Yaskawa INFORM job: A_ROOF_SIDE_0617_2_PAINT_46.JBI

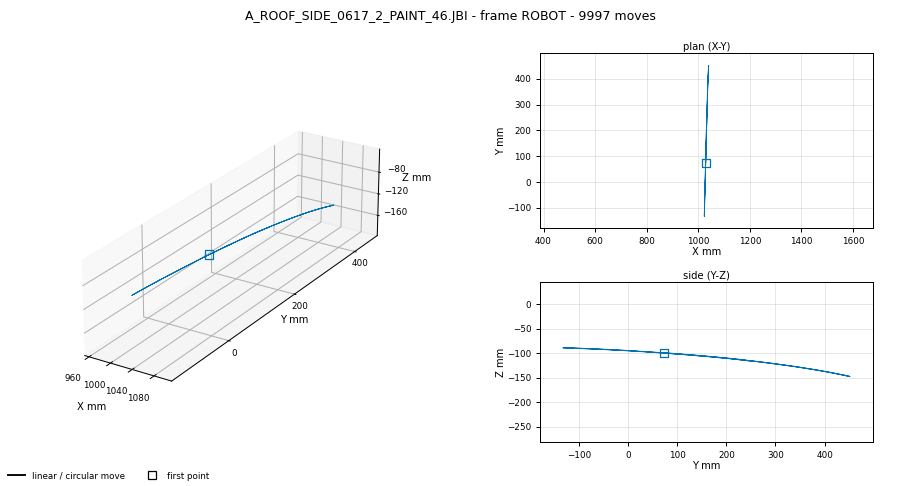
[picture p0: tool path of A_ROOF_SIDE_0617_2_PAINT_46.JBI in frame ROBOT, 9997 of 9997 moves have a stored position in this frame; points joined in program order, loops and branches not executed]
/JOB
//NAME A_ROOF_SIDE_0617_2_PAINT46
//POS
///NPOS 9997,0,0,0,0,0
///TOOL 1
///USER 0
///POSTYPE ROBOT
///RECTAN
///RCONF 1,0,0,0,0,0,0,0,0,0,0,0,0,0,0,0,0,0,0,0,0,0,0,0
C00000=1029.053,72.292,-98.591,168.354,44.972,158.390
C00001=1029.059,72.542,-98.608,168.356,44.969,158.390
C00002=1029.064,72.791,-98.626,168.358,44.967,158.389
C00003=1029.071,73.040,-98.644,168.360,44.965,158.389
C00004=1029.078,73.289,-98.662,168.362,44.963,158.389
C00005=1029.083,73.538,-98.680,168.365,44.961,158.389
C00006=1029.089,73.788,-98.698,168.367,44.958,158.389
C00007=1029.095,74.038,-98.715,168.370,44.956,158.388
C00008=1029.101,74.286,-98.734,168.373,44.954,158.388
C00009=1029.108,74.536,-98.751,168.375,44.951,158.388
C00010=1029.114,74.785,-98.769,168.377,44.949,158.388
C00011=1029.119,75.016,-98.786,168.380,44.947,158.388
C00012=1029.126,75.246,-98.802,168.381,44.945,158.387
C00013=1029.131,75.476,-98.818,168.384,44.943,158.387
C00014=1029.136,75.706,-98.836,168.386,44.941,158.387
C00015=1029.143,75.937,-98.852,168.389,44.939,158.387
C00016=1029.148,76.166,-98.868,168.390,44.937,158.387
C00017=1029.154,76.397,-98.886,168.393,44.935,158.387
C00018=1029.160,76.627,-98.902,168.395,44.933,158.387
C00019=1029.166,76.877,-98.920,168.398,44.931,158.386
C00020=1029.172,77.126,-98.938,168.400,44.928,158.386
C00021=1029.178,77.375,-98.956,168.403,44.926,158.386
C00022=1029.184,77.624,-98.974,168.405,44.924,158.386
C00023=1029.190,77.874,-98.992,168.408,44.922,158.386
C00024=1029.196,78.123,-99.010,168.409,44.920,158.385
C00025=1029.202,78.372,-99.029,168.412,44.917,158.385
C00026=1029.208,78.622,-99.047,168.414,44.915,158.385
C00027=1029.215,78.871,-99.065,168.417,44.913,158.385
C00028=1029.220,79.120,-99.083,168.419,44.911,158.385
C00029=1029.227,79.369,-99.101,168.422,44.909,158.385
C00030=1029.233,79.619,-99.119,168.424,44.907,158.384
C00031=1029.238,79.868,-99.138,168.427,44.905,158.384
C00032=1029.244,80.118,-99.156,168.429,44.902,158.384
C00033=1029.250,80.367,-99.175,168.432,44.900,158.384
C00034=1029.257,80.616,-99.193,168.434,44.898,158.384
C00035=1029.262,80.865,-99.211,168.437,44.895,158.383
C00036=1029.269,81.114,-99.230,168.438,44.894,158.383
C00037=1029.275,81.364,-99.248,168.441,44.892,158.383
C00038=1029.281,81.613,-99.266,168.443,44.889,158.383
C00039=1029.288,81.863,-99.284,168.446,44.887,158.383
C00040=1029.293,82.111,-99.302,168.448,44.885,158.383
C00041=1029.299,82.361,-99.320,168.450,44.883,158.382
C00042=1029.305,82.610,-99.340,168.453,44.881,158.382
C00043=1029.312,82.859,-99.358,168.456,44.879,158.382
C00044=1029.317,83.108,-99.376,168.458,44.876,158.382
C00045=1029.324,83.357,-99.395,168.460,44.874,158.382
C00046=1029.330,83.607,-99.412,168.463,44.872,158.382
C00047=1029.336,83.856,-99.431,168.465,44.869,158.381
C00048=1029.343,84.105,-99.450,168.468,44.867,158.381
C00049=1029.348,84.354,-99.467,168.470,44.865,158.381
C00050=1029.354,84.604,-99.486,168.473,44.863,158.381
C00051=1029.361,84.853,-99.505,168.475,44.861,158.381
C00052=1029.366,85.103,-99.523,168.477,44.858,158.380
C00053=1029.373,85.352,-99.542,168.479,44.856,158.380
C00054=1029.379,85.601,-99.560,168.482,44.855,158.380
C00055=1029.385,85.850,-99.578,168.484,44.852,158.380
C00056=1029.391,86.099,-99.597,168.487,44.850,158.380
C00057=1029.397,86.348,-99.615,168.489,44.847,158.379
C00058=1029.404,86.598,-99.633,168.492,44.845,158.379
C00059=1029.410,86.847,-99.652,168.494,44.843,158.379
C00060=1029.416,87.096,-99.671,168.496,44.841,158.379
C00061=1029.422,87.346,-99.690,168.499,44.839,158.379
C00062=1029.428,87.595,-99.707,168.501,44.836,158.378
C00063=1029.434,87.844,-99.726,168.504,44.834,158.378
C00064=1029.441,88.093,-99.745,168.506,44.832,158.378
C00065=1029.447,88.343,-99.763,168.509,44.830,158.378
C00066=1029.453,88.592,-99.781,168.511,44.828,158.378
C00067=1029.459,88.841,-99.800,168.514,44.825,158.378
C00068=1029.466,89.090,-99.819,168.516,44.823,158.377
C00069=1029.472,89.340,-99.838,168.519,44.820,158.377
C00070=1029.478,89.589,-99.856,168.521,44.818,158.377
C00071=1029.484,89.838,-99.874,168.524,44.816,158.377
C00072=1029.490,90.087,-99.893,168.526,44.814,158.377
C00073=1029.496,90.336,-99.912,168.529,44.812,158.376
C00074=1029.502,90.585,-99.931,168.531,44.810,158.376
C00075=1029.508,90.835,-99.950,168.533,44.807,158.376
C00076=1029.514,91.084,-99.968,168.535,44.806,158.376
C00077=1029.520,91.334,-99.987,168.538,44.804,158.376
C00078=1029.526,91.583,-100.006,168.540,44.802,158.376
C00079=1029.533,91.868,-100.028,168.544,44.799,158.375
C00080=1029.540,92.153,-100.049,168.546,44.796,158.375
C00081=1029.547,92.438,-100.070,168.548,44.794,158.375
C00082=1029.554,92.723,-100.092,168.552,44.791,158.375
C00083=1029.560,92.973,-100.111,168.554,44.789,158.375
C00084=1029.566,93.222,-100.130,168.557,44.787,158.375
C00085=1029.572,93.470,-100.148,168.559,44.785,158.374
C00086=1029.578,93.720,-100.167,168.561,44.783,158.374
C00087=1029.584,93.969,-100.186,168.563,44.781,158.374
C00088=1029.590,94.218,-100.205,168.566,44.779,158.374
C00089=1029.596,94.467,-100.224,168.568,44.777,158.374
C00090=1029.602,94.717,-100.243,168.571,44.775,158.373
C00091=1029.608,94.966,-100.262,168.573,44.772,158.373
C00092=1029.615,95.215,-100.281,168.576,44.770,158.373
C00093=1029.621,95.464,-100.299,168.578,44.768,158.373
C00094=1029.627,95.714,-100.319,168.581,44.765,158.373
C00095=1029.633,95.963,-100.337,168.583,44.763,158.372
C00096=1029.639,96.212,-100.356,168.586,44.762,158.372
C00097=1029.645,96.461,-100.375,168.588,44.759,158.372
C00098=1029.651,96.711,-100.394,168.591,44.757,158.372
C00099=1029.657,96.960,-100.413,168.593,44.755,158.372
C00100=1029.664,97.209,-100.432,168.596,44.752,158.371
C00101=1029.669,97.459,-100.451,168.598,44.750,158.371
C00102=1029.676,97.707,-100.470,168.601,44.748,158.371
C00103=1029.682,97.956,-100.490,168.603,44.746,158.371
C00104=1029.688,98.206,-100.508,168.606,44.744,158.371
C00105=1029.694,98.455,-100.527,168.608,44.741,158.371
C00106=1029.700,98.704,-100.546,168.610,44.739,158.370
C00107=1029.706,98.954,-100.565,168.613,44.737,158.370
C00108=1029.712,99.203,-100.584,168.615,44.735,158.370
C00109=1029.719,99.452,-100.603,168.618,44.733,158.370
C00110=1029.725,99.701,-100.623,168.620,44.731,158.370
C00111=1029.731,99.950,-100.641,168.623,44.728,158.369
C00112=1029.737,100.199,-100.660,168.625,44.726,158.369
C00113=1029.743,100.449,-100.680,168.628,44.724,158.369
C00114=1029.748,100.698,-100.699,168.631,44.722,158.369
C00115=1029.755,100.947,-100.718,168.632,44.720,158.369
C00116=1029.761,101.196,-100.738,168.634,44.718,158.369
C00117=1029.766,101.445,-100.757,168.637,44.716,158.368
C00118=1029.773,101.694,-100.776,168.640,44.714,158.368
C00119=1029.779,101.943,-100.795,168.642,44.711,158.368
C00120=1029.785,102.193,-100.815,168.644,44.710,158.368
C00121=1029.791,102.442,-100.835,168.647,44.708,158.368
C00122=1029.798,102.691,-100.854,168.650,44.706,158.368
C00123=1029.803,102.941,-100.873,168.652,44.703,158.367
C00124=1029.809,103.190,-100.893,168.654,44.701,158.367
C00125=1029.816,103.439,-100.911,168.657,44.699,158.367
C00126=1029.821,103.688,-100.931,168.660,44.697,158.367
C00127=1029.827,103.937,-100.951,168.662,44.695,158.367
C00128=1029.833,104.186,-100.970,168.665,44.693,158.367
C00129=1029.840,104.436,-100.989,168.667,44.691,158.366
C00130=1029.846,104.684,-101.009,168.670,44.689,158.366
C00131=1029.851,104.934,-101.028,168.672,44.686,158.366
C00132=1029.857,105.183,-101.047,168.675,44.684,158.366
C00133=1029.864,105.432,-101.066,168.677,44.682,158.366
C00134=1029.870,105.682,-101.086,168.679,44.680,158.365
C00135=1029.876,105.931,-101.106,168.682,44.678,158.365
C00136=1029.882,106.180,-101.125,168.685,44.676,158.365
C00137=1029.888,106.429,-101.145,168.687,44.674,158.365
C00138=1029.894,106.678,-101.164,168.690,44.671,158.365
C00139=1029.900,106.928,-101.183,168.692,44.669,158.365
C00140=1029.906,107.176,-101.202,168.695,44.667,158.365
C00141=1029.912,107.425,-101.222,168.697,44.665,158.364
C00142=1029.919,107.675,-101.242,168.700,44.663,158.364
C00143=1029.926,107.960,-101.264,168.702,44.660,158.364
C00144=1029.932,108.245,-101.286,168.705,44.658,158.364
C00145=1029.939,108.530,-101.308,168.708,44.655,158.363
C00146=1029.947,108.815,-101.331,168.710,44.653,158.363
C00147=1029.953,109.064,-101.350,168.713,44.651,158.363
C00148=1029.959,109.313,-101.370,168.715,44.649,158.363
C00149=1029.964,109.563,-101.389,168.718,44.647,158.363
C00150=1029.971,109.811,-101.409,168.720,44.644,158.363
C00151=1029.977,110.061,-101.428,168.723,44.642,158.362
C00152=1029.983,110.310,-101.448,168.725,44.640,158.362
C00153=1029.989,110.560,-101.468,168.728,44.638,158.362
C00154=1029.995,110.808,-101.488,168.730,44.636,158.362
C00155=1030.001,111.058,-101.507,168.733,44.634,158.362
C00156=1030.007,111.307,-101.527,168.735,44.632,158.362
C00157=1030.013,111.556,-101.547,168.738,44.629,158.361
C00158=1030.020,111.805,-101.566,168.740,44.627,158.361
C00159=1030.026,112.054,-101.586,168.743,44.625,158.361
C00160=1030.032,112.303,-101.606,168.745,44.624,158.361
C00161=1030.038,112.553,-101.625,168.748,44.621,158.361
C00162=1030.044,112.802,-101.645,168.750,44.619,158.360
C00163=1030.050,113.051,-101.665,168.753,44.617,158.360
C00164=1030.056,113.300,-101.684,168.755,44.615,158.360
C00165=1030.061,113.549,-101.705,168.758,44.613,158.360
C00166=1030.068,113.799,-101.725,168.761,44.611,158.360
C00167=1030.074,114.048,-101.745,168.763,44.609,158.360
C00168=1030.079,114.297,-101.764,168.766,44.607,158.360
C00169=1030.085,114.546,-101.784,168.768,44.605,158.359
C00170=1030.091,114.795,-101.804,168.771,44.603,158.359
C00171=1030.097,115.044,-101.825,168.773,44.601,158.359
C00172=1030.103,115.293,-101.845,168.776,44.599,158.359
C00173=1030.109,115.542,-101.865,168.778,44.597,158.359
C00174=1030.115,115.791,-101.884,168.781,44.595,158.359
C00175=1030.121,116.040,-101.904,168.784,44.593,158.359
C00176=1030.127,116.290,-101.925,168.786,44.591,158.358
C00177=1030.133,116.539,-101.945,168.788,44.589,158.358
C00178=1030.139,116.788,-101.965,168.791,44.587,158.358
C00179=1030.145,117.037,-101.985,168.794,44.585,158.358
C00180=1030.151,117.286,-102.006,168.796,44.583,158.358
C00181=1030.156,117.536,-102.025,168.799,44.581,158.358
C00182=1030.162,117.785,-102.045,168.801,44.579,158.357
C00183=1030.168,118.033,-102.065,168.804,44.577,158.357
C00184=1030.175,118.283,-102.086,168.806,44.575,158.357
C00185=1030.181,118.532,-102.106,168.809,44.572,158.357
C00186=1030.186,118.781,-102.126,168.811,44.570,158.357
C00187=1030.192,119.030,-102.146,168.814,44.568,158.357
C00188=1030.199,119.279,-102.166,168.817,44.567,158.357
C00189=1030.205,119.528,-102.186,168.819,44.565,158.356
C00190=1030.210,119.777,-102.207,168.822,44.563,158.356
C00191=1030.216,120.027,-102.227,168.824,44.561,158.356
C00192=1030.222,120.275,-102.247,168.827,44.558,158.356
C00193=1030.228,120.524,-102.267,168.829,44.556,158.356
C00194=1030.234,120.773,-102.287,168.832,44.554,158.356
C00195=1030.240,121.023,-102.308,168.834,44.552,158.355
C00196=1030.246,121.272,-102.328,168.837,44.550,158.355
C00197=1030.252,121.521,-102.348,168.839,44.548,158.355
C00198=1030.259,121.770,-102.368,168.842,44.546,158.355
C00199=1030.264,122.019,-102.389,168.844,44.544,158.355
C00200=1030.270,122.268,-102.409,168.847,44.542,158.355
C00201=1030.277,122.518,-102.429,168.849,44.540,158.354
C00202=1030.283,122.766,-102.449,168.852,44.538,158.354
C00203=1030.289,123.015,-102.469,168.855,44.536,158.354
C00204=1030.295,123.265,-102.490,168.857,44.534,158.354
C00205=1030.300,123.514,-102.510,168.860,44.532,158.354
C00206=1030.307,123.763,-102.530,168.862,44.530,158.354
C00207=1030.313,124.048,-102.554,168.865,44.527,158.353
C00208=1030.321,124.333,-102.577,168.868,44.525,158.353
C00209=1030.328,124.618,-102.600,168.871,44.522,158.353
C00210=1030.335,124.903,-102.624,168.874,44.520,158.353
C00211=1030.341,125.152,-102.644,168.877,44.518,158.353
C00212=1030.347,125.401,-102.663,168.879,44.516,158.353
C00213=1030.353,125.650,-102.684,168.881,44.514,158.352
C00214=1030.359,125.899,-102.704,168.885,44.512,158.352
C00215=1030.365,126.149,-102.725,168.888,44.510,158.352
C00216=1030.371,126.398,-102.745,168.890,44.508,158.352
C00217=1030.378,126.647,-102.766,168.893,44.506,158.352
C00218=1030.383,126.896,-102.786,168.895,44.503,158.352
C00219=1030.389,127.145,-102.806,168.898,44.501,158.351
C00220=1030.396,127.394,-102.827,168.900,44.499,158.351
C00221=1030.402,127.643,-102.846,168.903,44.497,158.351
C00222=1030.408,127.893,-102.867,168.905,44.496,158.351
C00223=1030.414,128.141,-102.888,168.908,44.493,158.351
C00224=1030.421,128.390,-102.908,168.910,44.491,158.351
C00225=1030.427,128.639,-102.928,168.913,44.489,158.350
C00226=1030.432,128.889,-102.949,168.916,44.487,158.350
C00227=1030.439,129.137,-102.970,168.919,44.485,158.350
C00228=1030.445,129.387,-102.990,168.921,44.482,158.350
C00229=1030.451,129.636,-103.010,168.924,44.481,158.350
C00230=1030.457,129.885,-103.031,168.927,44.479,158.350
C00231=1030.463,130.134,-103.051,168.929,44.477,158.350
C00232=1030.470,130.383,-103.072,168.931,44.474,158.349
C00233=1030.475,130.632,-103.093,168.934,44.472,158.349
C00234=1030.482,130.882,-103.113,168.937,44.470,158.349
C00235=1030.487,131.130,-103.134,168.939,44.468,158.349
C00236=1030.493,131.379,-103.154,168.942,44.466,158.349
C00237=1030.500,131.628,-103.176,168.945,44.464,158.349
C00238=1030.506,131.877,-103.196,168.948,44.462,158.348
C00239=1030.511,132.127,-103.217,168.951,44.460,158.348
C00240=1030.517,132.375,-103.238,168.953,44.458,158.348
C00241=1030.524,132.625,-103.258,168.956,44.457,158.348
C00242=1030.529,132.873,-103.280,168.958,44.455,158.348
C00243=1030.536,133.123,-103.300,168.961,44.453,158.348
C00244=1030.541,133.371,-103.321,168.963,44.451,158.348
C00245=1030.547,133.621,-103.342,168.966,44.449,158.347
C00246=1030.554,133.869,-103.363,168.969,44.447,158.347
C00247=1030.559,134.119,-103.384,168.971,44.445,158.347
C00248=1030.566,134.367,-103.404,168.973,44.442,158.347
C00249=1030.572,134.617,-103.425,168.976,44.440,158.347
C00250=1030.578,134.865,-103.446,168.980,44.438,158.347
C00251=1030.584,135.115,-103.467,168.982,44.436,158.347
C00252=1030.589,135.364,-103.488,168.985,44.434,158.346
C00253=1030.596,135.613,-103.509,168.987,44.433,158.346
C00254=1030.602,135.863,-103.530,168.990,44.431,158.346
C00255=1030.608,136.111,-103.550,168.993,44.429,158.346
C00256=1030.614,136.361,-103.572,168.995,44.427,158.346
C00257=1030.619,136.610,-103.592,168.998,44.425,158.346
C00258=1030.626,136.859,-103.613,169.000,44.423,158.346
C00259=1030.632,137.107,-103.635,169.003,44.421,158.345
C00260=1030.638,137.357,-103.656,169.006,44.419,158.345
C00261=1030.644,137.605,-103.676,169.009,44.417,158.345
C00262=1030.650,137.855,-103.697,169.012,44.415,158.345
C00263=1030.656,138.104,-103.719,169.014,44.413,158.345
C00264=1030.662,138.352,-103.739,169.017,44.411,158.345
C00265=1030.668,138.602,-103.760,169.019,44.409,158.345
C00266=1030.674,138.851,-103.782,169.022,44.407,158.344
C00267=1030.680,139.100,-103.803,169.024,44.405,158.344
C00268=1030.686,139.350,-103.824,169.027,44.404,158.344
C00269=1030.692,139.598,-103.845,169.031,44.401,158.344
C00270=1030.698,139.847,-103.867,169.033,44.399,158.344
C00271=1030.705,140.133,-103.891,169.036,44.398,158.344
C00272=1030.711,140.417,-103.915,169.039,44.395,158.344
C00273=1030.719,140.702,-103.939,169.042,44.393,158.343
C00274=1030.725,140.987,-103.964,169.045,44.391,158.343
C00275=1030.731,141.235,-103.985,169.048,44.389,158.343
C00276=1030.737,141.485,-104.006,169.050,44.387,158.343
C00277=1030.743,141.734,-104.027,169.053,44.385,158.343
C00278=1030.749,141.982,-104.049,169.056,44.383,158.343
C00279=1030.755,142.232,-104.070,169.059,44.381,158.343
C00280=1030.761,142.480,-104.092,169.062,44.379,158.343
C00281=1030.767,142.730,-104.112,169.064,44.377,158.342
C00282=1030.774,142.979,-104.133,169.067,44.375,158.342
C00283=1030.779,143.227,-104.155,169.069,44.373,158.342
C00284=1030.785,143.477,-104.176,169.072,44.371,158.342
C00285=1030.791,143.726,-104.198,169.075,44.369,158.342
C00286=1030.797,143.974,-104.219,169.078,44.367,158.342
C00287=1030.803,144.224,-104.240,169.081,44.365,158.342
C00288=1030.809,144.473,-104.262,169.083,44.363,158.341
C00289=1030.815,144.721,-104.283,169.086,44.362,158.341
C00290=1030.821,144.971,-104.304,169.089,44.360,158.341
C00291=1030.828,145.220,-104.326,169.091,44.358,158.341
C00292=1030.833,145.468,-104.347,169.094,44.356,158.341
C00293=1030.839,145.718,-104.369,169.097,44.354,158.341
C00294=1030.845,145.967,-104.390,169.100,44.352,158.341
C00295=1030.852,146.216,-104.412,169.103,44.351,158.341
C00296=1030.858,146.464,-104.433,169.105,44.349,158.341
C00297=1030.863,146.714,-104.455,169.108,44.347,158.340
C00298=1030.870,146.963,-104.476,169.110,44.345,158.340
C00299=1030.876,147.212,-104.498,169.114,44.343,158.340
C00300=1030.881,147.461,-104.519,169.117,44.341,158.340
C00301=1030.887,147.710,-104.541,169.119,44.339,158.340
C00302=1030.894,147.959,-104.563,169.122,44.337,158.340
C00303=1030.899,148.208,-104.584,169.124,44.335,158.340
C00304=1030.905,148.457,-104.606,169.127,44.333,158.339
C00305=1030.911,148.706,-104.627,169.131,44.332,158.340
C00306=1030.918,148.955,-104.649,169.133,44.330,158.339
C00307=1030.923,149.204,-104.670,169.136,44.328,158.339
C00308=1030.929,149.453,-104.692,169.138,44.326,158.339
C00309=1030.936,149.701,-104.714,169.141,44.324,158.339
C00310=1030.942,149.951,-104.736,169.144,44.322,158.339
C00311=1030.947,150.200,-104.758,169.147,44.320,158.339
C00312=1030.953,150.449,-104.779,169.150,44.319,158.339
C00313=1030.959,150.698,-104.801,169.153,44.317,158.339
C00314=1030.965,150.947,-104.823,169.155,44.315,158.338
C00315=1030.971,151.196,-104.844,169.158,44.313,158.338
C00316=1030.977,151.444,-104.866,169.161,44.311,158.338
C00317=1030.984,151.693,-104.888,169.164,44.309,158.338
C00318=1030.990,151.943,-104.909,169.167,44.308,158.338
C00319=1030.995,152.192,-104.932,169.169,44.306,158.338
C00320=1031.001,152.440,-104.954,169.172,44.304,158.338
C00321=1031.007,152.689,-104.975,169.176,44.302,158.338
C00322=1031.013,152.938,-104.997,169.178,44.300,158.338
C00323=1031.019,153.188,-105.019,169.181,44.298,158.337
C00324=1031.026,153.437,-105.040,169.183,44.296,158.337
C00325=1031.031,153.685,-105.062,169.186,44.295,158.337
C00326=1031.037,153.934,-105.084,169.190,44.293,158.337
C00327=1031.043,154.183,-105.106,169.192,44.291,158.337
C00328=1031.050,154.432,-105.128,169.195,44.289,158.337
C00329=1031.055,154.682,-105.151,169.197,44.287,158.337
C00330=1031.061,154.931,-105.172,169.200,44.286,158.337
C00331=1031.067,155.179,-105.194,169.204,44.284,158.337
C00332=1031.073,155.428,-105.216,169.206,44.282,158.336
C00333=1031.079,155.677,-105.238,169.209,44.280,158.336
C00334=1031.085,155.926,-105.260,169.212,44.279,158.336
C00335=1031.092,156.211,-105.285,169.215,44.276,158.336
C00336=1031.099,156.495,-105.311,169.219,44.274,158.336
C00337=1031.106,156.780,-105.336,169.222,44.272,158.336
C00338=1031.112,157.064,-105.361,169.225,44.270,158.336
C00339=1031.119,157.313,-105.383,169.228,44.268,158.336
C00340=1031.124,157.562,-105.405,169.230,44.266,158.336
C00341=1031.130,157.811,-105.428,169.234,44.264,158.336
C00342=1031.137,158.060,-105.449,169.236,44.262,158.335
C00343=1031.142,158.309,-105.472,169.239,44.261,158.335
C00344=1031.149,158.558,-105.494,169.242,44.259,158.335
C00345=1031.155,158.807,-105.516,169.245,44.257,158.335
C00346=1031.161,159.056,-105.538,169.248,44.255,158.335
C00347=1031.167,159.305,-105.560,169.251,44.254,158.335
C00348=1031.173,159.554,-105.582,169.253,44.252,158.335
C00349=1031.178,159.802,-105.605,169.257,44.250,158.335
C00350=1031.184,160.051,-105.627,169.260,44.249,158.335
C00351=1031.190,160.300,-105.650,169.262,44.247,158.335
C00352=1031.196,160.550,-105.672,169.265,44.246,158.335
C00353=1031.201,160.799,-105.695,169.268,44.244,158.334
C00354=1031.208,161.047,-105.717,169.271,44.242,158.334
C00355=1031.213,161.296,-105.740,169.274,44.240,158.334
C00356=1031.219,161.546,-105.762,169.277,44.238,158.334
C00357=1031.225,161.794,-105.785,169.280,44.237,158.334
C00358=1031.230,162.042,-105.807,169.282,44.235,158.334
C00359=1031.236,162.292,-105.829,169.286,44.234,158.334
C00360=1031.242,162.541,-105.852,169.289,44.232,158.334
C00361=1031.248,162.789,-105.875,169.291,44.231,158.334
C00362=1031.254,163.038,-105.898,169.294,44.229,158.334
C00363=1031.260,163.287,-105.921,169.298,44.227,158.334
C00364=1031.265,163.537,-105.943,169.300,44.225,158.334
C00365=1031.271,163.785,-105.965,169.303,44.224,158.334
C00366=1031.277,164.034,-105.988,169.306,44.222,158.334
C00367=1031.283,164.283,-106.011,169.308,44.220,158.333
C00368=1031.289,164.532,-106.034,169.312,44.219,158.334
C00369=1031.295,164.781,-106.056,169.315,44.217,158.333
C00370=1031.301,165.030,-106.079,169.318,44.216,158.333
C00371=1031.306,165.279,-106.102,169.320,44.214,158.333
C00372=1031.312,165.528,-106.125,169.324,44.212,158.333
C00373=1031.318,165.776,-106.147,169.327,44.211,158.333
C00374=1031.324,166.025,-106.170,169.329,44.209,158.333
C00375=1031.330,166.274,-106.193,169.333,44.207,158.333
C00376=1031.335,166.524,-106.215,169.336,44.206,158.333
C00377=1031.342,166.772,-106.237,169.338,44.204,158.333
C00378=1031.348,167.021,-106.260,169.341,44.203,158.333
C00379=1031.353,167.270,-106.283,169.345,44.201,158.333
C00380=1031.359,167.519,-106.306,169.348,44.199,158.333
C00381=1031.365,167.768,-106.329,169.350,44.198,158.333
C00382=1031.371,168.017,-106.352,169.354,44.195,158.333
C00383=1031.377,168.265,-106.374,169.357,44.194,158.333
C00384=1031.383,168.514,-106.397,169.359,44.192,158.332
C00385=1031.388,168.763,-106.420,169.362,44.191,158.332
C00386=1031.395,169.012,-106.443,169.366,44.189,158.332
C00387=1031.401,169.261,-106.466,169.368,44.188,158.332
C00388=1031.406,169.510,-106.489,169.371,44.186,158.332
C00389=1031.412,169.758,-106.512,169.375,44.184,158.332
C00390=1031.419,170.007,-106.534,169.377,44.182,158.332
C00391=1031.424,170.256,-106.557,169.380,44.181,158.332
C00392=1031.431,170.506,-106.580,169.384,44.179,158.332
C00393=1031.436,170.754,-106.603,169.387,44.178,158.332
C00394=1031.443,171.003,-106.625,169.389,44.176,158.332
C00395=1031.449,171.252,-106.648,169.393,44.175,158.332
C00396=1031.454,171.501,-106.671,169.396,44.173,158.332
C00397=1031.460,171.750,-106.694,169.398,44.171,158.332
C00398=1031.466,171.999,-106.717,169.402,44.169,158.332
C00399=1031.473,172.282,-106.744,169.406,44.167,158.332
C00400=1031.480,172.567,-106.769,169.408,44.166,158.332
C00401=1031.487,172.851,-106.796,169.412,44.164,158.331
C00402=1031.494,173.135,-106.822,169.416,44.162,158.331
C00403=1031.500,173.383,-106.845,169.418,44.161,158.331
C00404=1031.506,173.632,-106.868,169.422,44.158,158.331
C00405=1031.512,173.882,-106.891,169.425,44.157,158.331
C00406=1031.518,174.131,-106.914,169.428,44.155,158.331
C00407=1031.524,174.379,-106.937,169.431,44.154,158.331
C00408=1031.530,174.628,-106.960,169.434,44.152,158.331
C00409=1031.536,174.877,-106.983,169.438,44.151,158.331
C00410=1031.542,175.126,-107.007,169.440,44.149,158.331
C00411=1031.548,175.375,-107.029,169.444,44.147,158.331
C00412=1031.554,175.624,-107.052,169.447,44.145,158.331
C00413=1031.561,175.872,-107.075,169.449,44.144,158.331
C00414=1031.566,176.121,-107.098,169.453,44.142,158.331
C00415=1031.573,176.370,-107.122,169.456,44.141,158.331
C00416=1031.578,176.619,-107.145,169.459,44.139,158.331
C00417=1031.584,176.868,-107.168,169.462,44.137,158.331
C00418=1031.591,177.116,-107.191,169.465,44.136,158.330
C00419=1031.597,177.366,-107.214,169.469,44.134,158.331
C00420=1031.603,177.614,-107.238,169.471,44.132,158.330
C00421=1031.609,177.863,-107.261,169.475,44.131,158.330
C00422=1031.615,178.113,-107.284,169.478,44.130,158.330
C00423=1031.622,178.361,-107.306,169.481,44.127,158.330
C00424=1031.628,178.609,-107.330,169.484,44.126,158.330
C00425=1031.633,178.858,-107.353,169.488,44.124,158.330
C00426=1031.640,179.107,-107.377,169.491,44.123,158.330
C00427=1031.646,179.356,-107.400,169.493,44.121,158.330
C00428=1031.652,179.605,-107.423,169.497,44.120,158.330
C00429=1031.659,179.854,-107.446,169.500,44.118,158.330
C00430=1031.665,180.103,-107.469,169.504,44.116,158.330
C00431=1031.670,180.352,-107.492,169.506,44.114,158.330
C00432=1031.677,180.601,-107.516,169.510,44.113,158.330
C00433=1031.683,180.849,-107.539,169.513,44.111,158.330
C00434=1031.689,181.098,-107.563,169.516,44.110,158.330
C00435=1031.696,181.347,-107.585,169.519,44.108,158.330
C00436=1031.702,181.595,-107.609,169.523,44.106,158.330
C00437=1031.708,181.845,-107.632,169.526,44.105,158.330
C00438=1031.714,182.093,-107.656,169.529,44.103,158.330
C00439=1031.720,182.342,-107.679,169.532,44.102,158.330
C00440=1031.726,182.592,-107.702,169.536,44.100,158.329
C00441=1031.733,182.840,-107.725,169.538,44.098,158.329
C00442=1031.740,183.089,-107.749,169.542,44.097,158.330
C00443=1031.745,183.338,-107.773,169.545,44.095,158.329
C00444=1031.751,183.586,-107.797,169.549,44.094,158.329
C00445=1031.757,183.835,-107.821,169.551,44.092,158.329
C00446=1031.762,184.084,-107.844,169.554,44.091,158.329
C00447=1031.768,184.333,-107.869,169.558,44.090,158.329
C00448=1031.774,184.582,-107.893,169.561,44.088,158.329
C00449=1031.780,184.830,-107.916,169.565,44.087,158.330
C00450=1031.785,185.079,-107.940,169.568,44.086,158.330
C00451=1031.792,185.328,-107.964,169.570,44.084,158.329
C00452=1031.797,185.577,-107.988,169.574,44.082,158.329
C00453=1031.803,185.825,-108.012,169.577,44.081,158.329
C00454=1031.809,186.074,-108.036,169.581,44.080,158.329
C00455=1031.815,186.323,-108.060,169.583,44.079,158.329
C00456=1031.821,186.572,-108.083,169.587,44.077,158.330
C00457=1031.827,186.821,-108.108,169.590,44.076,158.330
C00458=1031.833,187.069,-108.131,169.594,44.074,158.330
C00459=1031.839,187.318,-108.156,169.597,44.073,158.330
C00460=1031.845,187.567,-108.179,169.601,44.072,158.330
C00461=1031.850,187.815,-108.204,169.603,44.070,158.329
C00462=1031.857,188.064,-108.228,169.607,44.068,158.329
C00463=1031.863,188.348,-108.255,169.611,44.067,158.330
C00464=1031.870,188.632,-108.282,169.614,44.066,158.330
C00465=1031.877,188.915,-108.310,169.617,44.064,158.330
C00466=1031.883,189.200,-108.337,169.621,44.062,158.329
C00467=1031.889,189.448,-108.361,169.625,44.061,158.330
C00468=1031.896,189.697,-108.385,169.628,44.060,158.330
C00469=1031.901,189.945,-108.409,169.631,44.058,158.330
C00470=1031.908,190.194,-108.433,169.634,44.057,158.330
C00471=1031.913,190.443,-108.457,169.638,44.056,158.330
C00472=1031.920,190.692,-108.481,169.642,44.054,158.330
C00473=1031.925,190.941,-108.506,169.645,44.053,158.330
C00474=1031.932,191.190,-108.530,169.649,44.051,158.330
C00475=1031.937,191.438,-108.554,169.651,44.050,158.330
C00476=1031.944,191.687,-108.578,169.655,44.049,158.330
C00477=1031.949,191.936,-108.602,169.658,44.048,158.330
C00478=1031.956,192.185,-108.626,169.662,44.046,158.330
C00479=1031.961,192.433,-108.651,169.665,44.045,158.330
C00480=1031.968,192.682,-108.675,169.668,44.043,158.330
C00481=1031.975,192.931,-108.699,169.671,44.042,158.330
C00482=1031.980,193.179,-108.724,169.675,44.041,158.330
C00483=1031.986,193.428,-108.748,169.678,44.040,158.330
C00484=1031.992,193.677,-108.772,169.682,44.038,158.330
C00485=1031.998,193.926,-108.796,169.686,44.037,158.330
C00486=1032.004,194.174,-108.820,169.688,44.035,158.330
C00487=1032.010,194.423,-108.844,169.692,44.034,158.330
C00488=1032.017,194.672,-108.869,169.695,44.033,158.330
C00489=1032.023,194.920,-108.893,169.699,44.031,158.330
C00490=1032.028,195.170,-108.918,169.703,44.030,158.330
C00491=1032.035,195.418,-108.941,169.705,44.029,158.330
C00492=1032.040,195.667,-108.966,169.709,44.027,158.330
C00493=1032.047,195.915,-108.991,169.712,44.026,158.330
C00494=1032.053,196.164,-109.015,169.716,44.025,158.330
C00495=1032.059,196.413,-109.039,169.720,44.023,158.330
C00496=1032.065,196.662,-109.064,169.723,44.022,158.330
C00497=1032.072,196.910,-109.088,169.726,44.020,158.330
C00498=1032.077,197.159,-109.113,169.729,44.019,158.330
C00499=1032.084,197.408,-109.137,169.733,44.018,158.330
C00500=1032.090,197.656,-109.162,169.737,44.016,158.330
C00501=1032.096,197.905,-109.186,169.740,44.015,158.330
C00502=1032.102,198.154,-109.210,169.744,44.014,158.330
C00503=1032.108,198.403,-109.234,169.747,44.012,158.330
C00504=1032.114,198.651,-109.259,169.750,44.011,158.330
C00505=1032.121,198.900,-109.283,169.754,44.010,158.330
C00506=1032.127,199.149,-109.309,169.758,44.008,158.330
C00507=1032.133,199.397,-109.332,169.761,44.007,158.330
C00508=1032.139,199.647,-109.357,169.764,44.006,158.331
C00509=1032.146,199.895,-109.382,169.768,44.004,158.331
C00510=1032.151,200.144,-109.406,169.771,44.003,158.331
C00511=1032.158,200.393,-109.430,169.775,44.001,158.331
C00512=1032.164,200.641,-109.455,169.779,44.000,158.331
C00513=1032.170,200.891,-109.480,169.782,43.999,158.331
C00514=1032.176,201.138,-109.505,169.786,43.998,158.331
C00515=1032.182,201.387,-109.530,169.788,43.997,158.331
C00516=1032.188,201.636,-109.555,169.792,43.995,158.331
C00517=1032.195,201.885,-109.580,169.796,43.995,158.331
C00518=1032.200,202.133,-109.604,169.799,43.993,158.331
C00519=1032.206,202.382,-109.629,169.803,43.992,158.331
C00520=1032.213,202.631,-109.655,169.807,43.991,158.331
C00521=1032.218,202.880,-109.679,169.810,43.990,158.331
C00522=1032.224,203.128,-109.704,169.814,43.989,158.331
C00523=1032.230,203.377,-109.730,169.817,43.987,158.331
C00524=1032.237,203.626,-109.754,169.820,43.987,158.331
C00525=1032.243,203.874,-109.779,169.824,43.985,158.332
C00526=1032.249,204.123,-109.804,169.828,43.984,158.332
C00527=1032.275,205.172,-109.909,170.170,44.088,158.383
C00528=1032.284,205.525,-109.947,170.174,44.087,158.384
C00529=1032.294,205.878,-109.984,170.178,44.087,158.384
C00530=1032.304,206.232,-110.022,170.181,44.087,158.384
C00531=1032.313,206.584,-110.058,170.185,44.086,158.384
C00532=1032.319,206.833,-110.085,170.187,44.085,158.384
C00533=1032.326,207.081,-110.111,170.190,44.085,158.384
C00534=1032.333,207.330,-110.138,170.192,44.084,158.385
C00535=1032.340,207.579,-110.164,170.195,44.084,158.385
C00536=1032.347,207.827,-110.190,170.197,44.084,158.385
C00537=1032.353,208.076,-110.217,170.200,44.083,158.385
C00538=1032.360,208.323,-110.244,170.202,44.083,158.385
C00539=1032.367,208.572,-110.270,170.205,44.082,158.385
C00540=1032.374,208.821,-110.297,170.208,44.082,158.385
C00541=1032.380,209.069,-110.323,170.211,44.082,158.386
C00542=1032.387,209.318,-110.350,170.214,44.082,158.386
C00543=1032.394,209.566,-110.376,170.216,44.081,158.386
C00544=1032.400,209.815,-110.403,170.219,44.081,158.386
C00545=1032.407,210.064,-110.429,170.221,44.080,158.386
C00546=1032.414,210.312,-110.455,170.224,44.080,158.387
C00547=1032.421,210.560,-110.482,170.226,44.080,158.387
C00548=1032.427,210.809,-110.510,170.229,44.079,158.387
C00549=1032.434,211.057,-110.536,170.231,44.079,158.387
C00550=1032.440,211.306,-110.563,170.235,44.079,158.387
C00551=1032.447,211.555,-110.589,170.237,44.078,158.387
C00552=1032.453,211.803,-110.616,170.240,44.078,158.387
C00553=1032.461,212.051,-110.643,170.242,44.077,158.387
C00554=1032.466,212.300,-110.669,170.245,44.077,158.388
C00555=1032.474,212.548,-110.697,170.248,44.077,158.388
C00556=1032.481,212.797,-110.723,170.250,44.076,158.388
C00557=1032.487,213.045,-110.750,170.253,44.077,158.388
C00558=1032.494,213.294,-110.776,170.255,44.076,158.388
C00559=1032.500,213.542,-110.804,170.258,44.076,158.389
C00560=1032.508,213.791,-110.830,170.261,44.076,158.389
C00561=1032.513,214.039,-110.857,170.264,44.075,158.389
C00562=1032.521,214.287,-110.884,170.266,44.075,158.389
C00563=1032.527,214.536,-110.911,170.269,44.074,158.389
C00564=1032.534,214.784,-110.937,170.272,44.074,158.389
C00565=1032.540,215.033,-110.965,170.274,44.074,158.390
C00566=1032.547,215.282,-110.991,170.277,44.073,158.390
C00567=1032.553,215.529,-111.019,170.279,44.073,158.390
C00568=1032.561,215.778,-111.045,170.282,44.073,158.390
C00569=1032.567,216.027,-111.072,170.284,44.072,158.390
C00570=1032.574,216.275,-111.099,170.288,44.073,158.391
C00571=1032.580,216.524,-111.126,170.291,44.072,158.391
C00572=1032.588,216.772,-111.153,170.293,44.072,158.391
C00573=1032.594,217.021,-111.180,170.296,44.072,158.391
C00574=1032.601,217.269,-111.207,170.298,44.071,158.391
C00575=1032.607,217.517,-111.234,170.301,44.071,158.391
C00576=1032.614,217.766,-111.260,170.304,44.070,158.391
C00577=1032.621,218.015,-111.288,170.306,44.070,158.392
C00578=1032.628,218.263,-111.314,170.309,44.070,158.392
C00579=1032.635,218.512,-111.342,170.312,44.069,158.392
C00580=1032.641,218.760,-111.368,170.315,44.069,158.392
C00581=1032.648,219.008,-111.396,170.318,44.069,158.392
C00582=1032.655,219.257,-111.422,170.320,44.068,158.392
C00583=1032.662,219.505,-111.450,170.323,44.068,158.393
C00584=1032.671,219.864,-111.489,170.327,44.067,158.393
C00585=1032.681,220.223,-111.529,170.331,44.067,158.393
C00586=1032.690,220.581,-111.568,170.335,44.067,158.394
C00587=1032.700,220.941,-111.608,170.339,44.067,158.394
C00588=1032.707,221.189,-111.635,170.342,44.067,158.394
C00589=1032.713,221.437,-111.662,170.344,44.066,158.394
C00590=1032.719,221.685,-111.689,170.347,44.066,158.394
C00591=1032.726,221.934,-111.717,170.350,44.066,158.395
C00592=1032.733,222.183,-111.743,170.352,44.066,158.395
C00593=1032.740,222.431,-111.771,170.355,44.065,158.395
C00594=1032.746,222.679,-111.798,170.358,44.065,158.395
C00595=1032.753,222.927,-111.826,170.361,44.065,158.395
C00596=1032.759,223.176,-111.853,170.364,44.064,158.396
C00597=1032.767,223.424,-111.880,170.366,44.065,158.396
C00598=1032.773,223.673,-111.908,170.369,44.064,158.396
C00599=1032.780,223.921,-111.936,170.372,44.064,158.396
C00600=1032.786,224.170,-111.963,170.374,44.064,158.396
C00601=1032.792,224.418,-111.990,170.378,44.064,158.397
C00602=1032.800,224.666,-112.017,170.381,44.063,158.397
C00603=1032.806,224.915,-112.045,170.383,44.063,158.397
C00604=1032.813,225.163,-112.073,170.386,44.063,158.397
C00605=1032.819,225.412,-112.100,170.389,44.063,158.397
C00606=1032.826,225.661,-112.128,170.391,44.062,158.398
C00607=1032.834,225.909,-112.155,170.394,44.062,158.398
C00608=1032.840,226.157,-112.182,170.398,44.062,158.398
C00609=1032.847,226.406,-112.210,170.400,44.061,158.398
C00610=1032.854,226.654,-112.238,170.403,44.061,158.398
C00611=1032.860,226.903,-112.266,170.406,44.061,158.399
C00612=1032.867,227.150,-112.292,170.408,44.061,158.399
C00613=1032.874,227.399,-112.319,170.411,44.060,158.399
C00614=1032.880,227.647,-112.347,170.415,44.060,158.399
C00615=1032.887,227.896,-112.375,170.418,44.060,158.399
C00616=1032.894,228.144,-112.403,170.420,44.060,158.400
C00617=1032.900,228.393,-112.430,170.423,44.060,158.400
C00618=1032.907,228.641,-112.458,170.426,44.060,158.400
C00619=1032.914,228.890,-112.486,170.428,44.060,158.400
C00620=1032.920,229.138,-112.514,170.431,44.059,158.400
C00621=1032.927,229.387,-112.541,170.435,44.059,158.401
C00622=1032.934,229.634,-112.570,170.437,44.059,158.401
C00623=1032.941,229.883,-112.597,170.440,44.059,158.401
C00624=1032.947,230.131,-112.625,170.443,44.059,158.401
C00625=1032.954,230.380,-112.653,170.445,44.059,158.401
C00626=1032.961,230.628,-112.681,170.449,44.059,158.402
C00627=1032.967,230.877,-112.708,170.452,44.058,158.402
C00628=1032.974,231.125,-112.736,170.454,44.058,158.402
C00629=1032.981,231.374,-112.764,170.457,44.058,158.402
C00630=1032.987,231.622,-112.792,170.460,44.058,158.403
C00631=1032.994,231.870,-112.821,170.463,44.058,158.403
C00632=1033.000,232.119,-112.848,170.466,44.058,158.403
C00633=1033.007,232.367,-112.876,170.469,44.057,158.403
C00634=1033.014,232.615,-112.904,170.472,44.057,158.404
C00635=1033.020,232.864,-112.932,170.474,44.058,158.404
C00636=1033.027,233.112,-112.961,170.477,44.057,158.404
C00637=1033.033,233.360,-112.988,170.481,44.057,158.404
C00638=1033.040,233.609,-113.016,170.484,44.057,158.405
C00639=1033.047,233.857,-113.044,170.486,44.057,158.405
C00640=1033.056,234.208,-113.084,170.490,44.056,158.405
C00641=1033.065,234.559,-113.123,170.494,44.056,158.405
C00642=1033.074,234.911,-113.163,170.499,44.056,158.406
C00643=1033.084,235.261,-113.202,170.503,44.056,158.406
C00644=1033.090,235.510,-113.231,170.506,44.056,158.406
C00645=1033.097,235.758,-113.259,170.508,44.056,158.407
C00646=1033.104,236.006,-113.287,170.512,44.056,158.407
C00647=1033.111,236.255,-113.316,170.515,44.056,158.407
C00648=1033.117,236.504,-113.344,170.518,44.056,158.407
C00649=1033.124,236.752,-113.372,170.520,44.056,158.408
C00650=1033.131,237.000,-113.400,170.523,44.055,158.408
C00651=1033.138,237.248,-113.428,170.527,44.055,158.408
C00652=1033.145,237.496,-113.456,170.530,44.055,158.408
C00653=1033.151,237.745,-113.485,170.532,44.055,158.408
C00654=1033.158,237.993,-113.513,170.535,44.055,158.409
C00655=1033.164,238.241,-113.541,170.538,44.055,158.409
C00656=1033.172,238.490,-113.569,170.542,44.055,158.409
C00657=1033.178,238.738,-113.598,170.545,44.055,158.409
C00658=1033.184,238.987,-113.626,170.547,44.055,158.410
C00659=1033.191,239.235,-113.654,170.550,44.055,158.410
C00660=1033.197,239.484,-113.683,170.554,44.055,158.410
C00661=1033.204,239.731,-113.711,170.557,44.054,158.410
C00662=1033.211,239.980,-113.739,170.560,44.054,158.411
C00663=1033.219,240.228,-113.767,170.562,44.055,158.411
C00664=1033.225,240.476,-113.797,170.565,44.055,158.411
C00665=1033.232,240.725,-113.824,170.569,44.055,158.412
C00666=1033.238,240.973,-113.853,170.572,44.054,158.412
C00667=1033.245,241.221,-113.882,170.574,44.054,158.412
C00668=1033.251,241.470,-113.910,170.577,44.054,158.412
C00669=1033.258,241.717,-113.939,170.580,44.054,158.413
C00670=1033.265,241.966,-113.968,170.584,44.054,158.413
C00671=1033.271,242.215,-113.996,170.587,44.054,158.413
C00672=1033.278,242.463,-114.025,170.589,44.055,158.413
C00673=1033.284,242.711,-114.054,170.593,44.055,158.414
C00674=1033.290,242.959,-114.081,170.596,44.055,158.414
C00675=1033.297,243.208,-114.111,170.599,44.054,158.414
C00676=1033.304,243.456,-114.139,170.602,44.054,158.414
C00677=1033.311,243.704,-114.168,170.605,44.054,158.415
C00678=1033.318,243.952,-114.197,170.608,44.054,158.415
C00679=1033.323,244.201,-114.225,170.611,44.054,158.415
C00680=1033.331,244.449,-114.254,170.614,44.054,158.416
C00681=1033.337,244.697,-114.283,170.617,44.054,158.416
C00682=1033.344,244.946,-114.312,170.621,44.054,158.416
C00683=1033.351,245.193,-114.340,170.623,44.055,158.416
C00684=1033.357,245.441,-114.370,170.626,44.055,158.417
C00685=1033.364,245.690,-114.399,170.630,44.055,158.417
C00686=1033.370,245.938,-114.428,170.633,44.055,158.417
C00687=1033.376,246.187,-114.457,170.636,44.055,158.418
C00688=1033.383,246.435,-114.485,170.638,44.055,158.418
C00689=1033.389,246.683,-114.514,170.642,44.055,158.418
C00690=1033.396,246.932,-114.543,170.645,44.055,158.418
C00691=1033.402,247.180,-114.572,170.648,44.055,158.419
C00692=1033.408,247.428,-114.601,170.651,44.055,158.419
C00693=1033.415,247.676,-114.630,170.655,44.055,158.419
C00694=1033.422,247.925,-114.659,170.657,44.055,158.420
C00695=1033.429,248.172,-114.689,170.660,44.055,158.420
C00696=1033.438,248.518,-114.729,170.665,44.056,158.420
C00697=1033.447,248.863,-114.770,170.669,44.056,158.421
C00698=1033.456,249.208,-114.810,170.673,44.056,158.421
C00699=1033.465,249.553,-114.850,170.678,44.056,158.422
C00700=1033.472,249.802,-114.880,170.681,44.056,158.422
C00701=1033.478,250.050,-114.909,170.684,44.056,158.422
C00702=1033.485,250.299,-114.938,170.688,44.057,158.423
C00703=1033.491,250.547,-114.967,170.691,44.057,158.423
C00704=1033.498,250.795,-114.997,170.693,44.057,158.423
C00705=1033.505,251.043,-115.025,170.697,44.057,158.423
C00706=1033.511,251.291,-115.054,170.700,44.057,158.424
C00707=1033.518,251.540,-115.084,170.703,44.057,158.424
C00708=1033.524,251.788,-115.113,170.706,44.057,158.424
C00709=1033.531,252.037,-115.142,170.710,44.057,158.425
C00710=1033.539,252.284,-115.171,170.713,44.057,158.425
C00711=1033.545,252.532,-115.200,170.716,44.057,158.425
C00712=1033.552,252.781,-115.230,170.720,44.058,158.426
C00713=1033.558,253.029,-115.259,170.723,44.058,158.426
C00714=1033.565,253.277,-115.289,170.725,44.058,158.426
C00715=1033.571,253.525,-115.318,170.729,44.058,158.426
C00716=1033.578,253.773,-115.346,170.732,44.058,158.427
C00717=1033.585,254.022,-115.376,170.735,44.058,158.427
C00718=1033.592,254.269,-115.406,170.738,44.058,158.427
C00719=1033.599,254.518,-115.435,170.742,44.058,158.428
C00720=1033.605,254.766,-115.464,170.745,44.058,158.428
C00721=1033.612,255.015,-115.494,170.748,44.059,158.428
C00722=1033.618,255.263,-115.523,170.752,44.059,158.429
C00723=1033.625,255.511,-115.552,170.755,44.059,158.429
C00724=1033.632,255.759,-115.582,170.758,44.059,158.429
C00725=1033.639,256.007,-115.611,170.761,44.059,158.430
C00726=1033.646,256.255,-115.641,170.765,44.059,158.430
C00727=1033.652,256.503,-115.670,170.768,44.059,158.430
C00728=1033.659,256.752,-115.699,170.771,44.060,158.431
C00729=1033.665,257.000,-115.729,170.775,44.060,158.431
C00730=1033.673,257.248,-115.758,170.778,44.060,158.431
C00731=1033.680,257.496,-115.788,170.781,44.060,158.431
C00732=1033.686,257.745,-115.817,170.785,44.060,158.432
C00733=1033.693,257.992,-115.847,170.788,44.060,158.432
C00734=1033.700,258.241,-115.876,170.791,44.061,158.433
C00735=1033.707,258.489,-115.906,170.795,44.061,158.433
C00736=1033.713,258.737,-115.935,170.798,44.061,158.433
C00737=1033.721,258.985,-115.965,170.801,44.061,158.433
C00738=1033.727,259.233,-115.994,170.804,44.061,158.434
C00739=1033.735,259.481,-116.024,170.808,44.061,158.434
C00740=1033.741,259.730,-116.053,170.811,44.061,158.434
C00741=1033.748,259.978,-116.083,170.814,44.061,158.435
C00742=1033.755,260.227,-116.113,170.818,44.061,158.435
C00743=1033.761,260.474,-116.142,170.821,44.061,158.435
C00744=1033.769,260.722,-116.173,170.824,44.062,158.436
C00745=1033.775,260.970,-116.201,170.828,44.062,158.436
C00746=1033.783,261.218,-116.231,170.831,44.062,158.436
C00747=1033.789,261.467,-116.261,170.834,44.062,158.437
C00748=1033.796,261.715,-116.290,170.838,44.063,158.437
C00749=1033.802,261.963,-116.321,170.841,44.063,158.437
C00750=1033.809,262.211,-116.351,170.844,44.063,158.438
C00751=1033.816,262.459,-116.381,170.848,44.064,158.438
C00752=1033.824,262.803,-116.422,170.852,44.064,158.439
C00753=1033.834,263.147,-116.464,170.857,44.064,158.439
C00754=1033.843,263.491,-116.505,170.861,44.065,158.440
C00755=1033.853,263.835,-116.547,170.867,44.065,158.440
C00756=1033.859,264.082,-116.577,170.870,44.065,158.441
C00757=1033.866,264.331,-116.607,170.873,44.065,158.441
C00758=1033.873,264.579,-116.638,170.877,44.066,158.441
C00759=1033.879,264.827,-116.667,170.880,44.066,158.442
C00760=1033.886,265.075,-116.697,170.884,44.066,158.442
C00761=1033.893,265.324,-116.727,170.887,44.067,158.442
C00762=1033.899,265.571,-116.757,170.890,44.067,158.443
C00763=1033.907,265.819,-116.787,170.894,44.067,158.443
C00764=1033.914,266.068,-116.817,170.897,44.068,158.444
C00765=1033.920,266.315,-116.848,170.900,44.068,158.444
C00766=1033.927,266.564,-116.878,170.904,44.068,158.444
C00767=1033.934,266.812,-116.908,170.907,44.069,158.445
C00768=1033.940,267.060,-116.938,170.911,44.069,158.445
C00769=1033.947,267.308,-116.969,170.914,44.069,158.445
C00770=1033.953,267.556,-116.999,170.918,44.070,158.446
C00771=1033.960,267.803,-117.030,170.921,44.070,158.446
C00772=1033.967,268.051,-117.060,170.924,44.071,158.446
C00773=1033.974,268.300,-117.091,170.928,44.071,158.447
C00774=1033.981,268.548,-117.121,170.932,44.071,158.447
C00775=1033.987,268.796,-117.151,170.935,44.071,158.448
C00776=1033.994,269.044,-117.181,170.939,44.072,158.448
C00777=1034.001,269.292,-117.211,170.942,44.072,158.448
C00778=1034.007,269.540,-117.242,170.946,44.072,158.449
C00779=1034.014,269.788,-117.272,170.949,44.073,158.449
C00780=1034.021,270.036,-117.303,170.952,44.073,158.450
C00781=1034.028,270.285,-117.333,170.956,44.074,158.450
C00782=1034.034,270.532,-117.364,170.959,44.074,158.450
C00783=1034.041,270.780,-117.394,170.963,44.074,158.451
C00784=1034.048,271.029,-117.425,170.966,44.075,158.451
C00785=1034.055,271.277,-117.455,170.970,44.075,158.452
C00786=1034.061,271.524,-117.486,170.974,44.075,158.452
C00787=1034.068,271.772,-117.517,170.977,44.076,158.452
C00788=1034.074,272.021,-117.547,170.981,44.076,158.453
C00789=1034.081,272.269,-117.579,170.984,44.077,158.453
C00790=1034.088,272.517,-117.609,170.988,44.077,158.454
C00791=1034.094,272.765,-117.639,170.991,44.077,158.454
C00792=1034.102,273.012,-117.670,170.995,44.078,158.454
C00793=1034.108,273.261,-117.701,170.998,44.079,158.455
C00794=1034.115,273.509,-117.732,171.002,44.078,158.455
C00795=1034.122,273.757,-117.762,171.006,44.079,158.456
C00796=1034.129,274.005,-117.794,171.009,44.080,158.456
C00797=1034.134,274.253,-117.824,171.013,44.080,158.457
C00798=1034.142,274.500,-117.855,171.016,44.080,158.457
C00799=1034.148,274.749,-117.886,171.020,44.081,158.457
C00800=1034.155,274.997,-117.917,171.023,44.082,158.458
C00801=1034.162,275.245,-117.947,171.028,44.082,158.458
C00802=1034.169,275.493,-117.979,171.031,44.083,158.459
C00803=1034.175,275.741,-118.009,171.034,44.083,158.459
C00804=1034.182,275.988,-118.040,171.038,44.083,158.459
C00805=1034.189,276.237,-118.070,171.041,44.084,158.460
C00806=1034.195,276.485,-118.102,171.045,44.085,158.460
C00807=1034.203,276.732,-118.133,171.048,44.085,158.461
C00808=1034.212,277.081,-118.176,171.054,44.086,158.461
C00809=1034.221,277.429,-118.219,171.059,44.087,158.462
C00810=1034.231,277.778,-118.263,171.064,44.087,158.463
C00811=1034.240,278.127,-118.307,171.069,44.088,158.463
C00812=1034.247,278.375,-118.338,171.073,44.088,158.464
C00813=1034.254,278.623,-118.370,171.077,44.089,158.464
C00814=1034.261,278.870,-118.401,171.080,44.090,158.465
C00815=1034.267,279.118,-118.433,171.084,44.090,158.465
C00816=1034.274,279.367,-118.463,171.087,44.090,158.465
C00817=1034.281,279.614,-118.494,171.091,44.091,158.466
C00818=1034.287,279.862,-118.525,171.095,44.091,158.466
C00819=1034.294,280.110,-118.557,171.099,44.092,158.467
C00820=1034.301,280.358,-118.588,171.102,44.093,158.467
C00821=1034.308,280.605,-118.619,171.106,44.093,158.468
C00822=1034.314,280.853,-118.651,171.109,44.094,158.468
C00823=1034.321,281.101,-118.682,171.114,44.094,158.469
C00824=1034.327,281.350,-118.713,171.117,44.095,158.469
C00825=1034.334,281.598,-118.744,171.121,44.096,158.470
C00826=1034.341,281.846,-118.776,171.124,44.096,158.470
C00827=1034.348,282.093,-118.807,171.128,44.097,158.470
C00828=1034.354,282.341,-118.839,171.132,44.097,158.471
C00829=1034.361,282.589,-118.870,171.136,44.098,158.471
C00830=1034.368,282.837,-118.902,171.139,44.099,158.472
C00831=1034.374,283.085,-118.933,171.143,44.099,158.472
C00832=1034.381,283.333,-118.964,171.147,44.100,158.473
C00833=1034.389,283.582,-118.996,171.151,44.100,158.473
C00834=1034.395,283.829,-119.028,171.154,44.101,158.474
C00835=1034.402,284.077,-119.060,171.158,44.102,158.474
C00836=1034.410,284.324,-119.091,171.163,44.103,158.475
C00837=1034.416,284.572,-119.122,171.166,44.103,158.475
C00838=1034.423,284.820,-119.154,171.170,44.104,158.476
C00839=1034.430,285.068,-119.185,171.174,44.104,158.476
C00840=1034.437,285.316,-119.216,171.178,44.105,158.477
C00841=1034.443,285.564,-119.248,171.181,44.106,158.477
C00842=1034.450,285.812,-119.279,171.185,44.106,158.478
C00843=1034.458,286.060,-119.312,171.189,44.107,158.478
C00844=1034.464,286.308,-119.343,171.193,44.107,158.479
C00845=1034.471,286.556,-119.375,171.196,44.108,158.479
C00846=1034.478,286.803,-119.406,171.201,44.109,158.480
C00847=1034.484,287.051,-119.439,171.204,44.110,158.480
C00848=1034.491,287.299,-119.470,171.208,44.110,158.481
C00849=1034.498,287.547,-119.502,171.211,44.111,158.481
C00850=1034.505,287.795,-119.534,171.216,44.111,158.481
C00851=1034.512,288.043,-119.566,171.220,44.113,158.482
C00852=1034.518,288.291,-119.598,171.223,44.113,158.483
C00853=1034.525,288.538,-119.630,171.228,44.114,158.483
C00854=1034.532,288.786,-119.661,171.231,44.114,158.483
C00855=1034.539,289.033,-119.693,171.235,44.116,158.484
C00856=1034.546,289.282,-119.725,171.239,44.116,158.485
C00857=1034.552,289.530,-119.758,171.243,44.117,158.485
C00858=1034.559,289.778,-119.789,171.247,44.118,158.486
C00859=1034.566,290.025,-119.822,171.251,44.118,158.486
C00860=1034.573,290.273,-119.853,171.255,44.119,158.487
C00861=1034.580,290.521,-119.886,171.258,44.120,158.487
C00862=1034.587,290.769,-119.918,171.263,44.121,158.488
C00863=1034.594,291.016,-119.950,171.266,44.121,158.488
C00864=1034.604,291.377,-119.996,171.272,44.123,158.489
C00865=1034.613,291.737,-120.043,171.278,44.123,158.490
C00866=1034.623,292.098,-120.089,171.284,44.124,158.490
C00867=1034.634,292.458,-120.137,171.289,44.126,158.491
C00868=1034.640,292.706,-120.168,171.294,44.126,158.492
C00869=1034.647,292.955,-120.201,171.297,44.128,158.492
C00870=1034.654,293.202,-120.233,171.302,44.128,158.493
C00871=1034.660,293.450,-120.265,171.306,44.129,158.494
C00872=1034.667,293.697,-120.297,171.309,44.130,158.494
C00873=1034.675,293.945,-120.330,171.314,44.130,158.494
C00874=1034.681,294.193,-120.363,171.317,44.132,158.495
C00875=1034.688,294.441,-120.394,171.321,44.132,158.496
C00876=1034.695,294.689,-120.427,171.326,44.133,158.496
C00877=1034.702,294.936,-120.459,171.329,44.134,158.497
C00878=1034.708,295.184,-120.492,171.334,44.135,158.497
C00879=1034.716,295.432,-120.525,171.338,44.136,158.498
C00880=1034.722,295.680,-120.557,171.341,44.137,158.498
C00881=1034.728,295.927,-120.590,171.346,44.138,158.499
C00882=1034.735,296.176,-120.623,171.350,44.139,158.500
C00883=1034.742,296.423,-120.655,171.353,44.140,158.500
C00884=1034.748,296.670,-120.688,171.358,44.141,158.501
C00885=1034.755,296.919,-120.721,171.362,44.142,158.501
C00886=1034.762,297.166,-120.753,171.366,44.142,158.502
C00887=1034.769,297.414,-120.786,171.370,44.144,158.502
C00888=1034.776,297.662,-120.819,171.374,44.145,158.503
C00889=1034.782,297.909,-120.852,171.378,44.145,158.504
C00890=1034.789,298.157,-120.884,171.382,44.147,158.504
C00891=1034.796,298.405,-120.917,171.387,44.148,158.505
C00892=1034.802,298.652,-120.951,171.390,44.148,158.505
C00893=1034.809,298.900,-120.984,171.394,44.149,158.506
C00894=1034.816,299.148,-121.016,171.399,44.150,158.507
C00895=1034.823,299.395,-121.049,171.402,44.152,158.507
C00896=1034.830,299.643,-121.082,171.407,44.152,158.508
C00897=1034.836,299.891,-121.115,171.411,44.153,158.508
C00898=1034.844,300.138,-121.148,171.415,44.154,158.509
C00899=1034.850,300.386,-121.180,171.419,44.156,158.510
C00900=1034.857,300.634,-121.214,171.424,44.156,158.510
C00901=1034.863,300.882,-121.246,171.427,44.157,158.511
C00902=1034.871,301.129,-121.280,171.431,44.159,158.511
C00903=1034.877,301.377,-121.312,171.436,44.160,158.512
C00904=1034.884,301.625,-121.345,171.440,44.161,158.513
C00905=1034.891,301.872,-121.379,171.444,44.161,158.513
C00906=1034.899,302.120,-121.411,171.448,44.162,158.514
C00907=1034.905,302.368,-121.444,171.453,44.163,158.514
C00908=1034.912,302.615,-121.478,171.456,44.165,158.515
C00909=1034.918,302.863,-121.511,171.461,44.166,158.516
C00910=1034.926,303.111,-121.543,171.465,44.167,158.516
C00911=1034.933,303.358,-121.577,171.470,44.168,158.517
C00912=1034.940,303.606,-121.610,171.473,44.169,158.517
C00913=1034.946,303.853,-121.643,171.478,44.170,158.518
C00914=1034.954,304.101,-121.676,171.482,44.171,158.519
C00915=1034.961,304.349,-121.710,171.486,44.172,158.519
C00916=1034.967,304.596,-121.742,171.490,44.173,158.520
C00917=1034.974,304.844,-121.776,171.495,44.174,158.521
C00918=1034.981,305.092,-121.809,171.500,44.175,158.521
C00919=1034.989,305.339,-121.842,171.503,44.176,158.522
C00920=1034.999,305.717,-121.893,171.510,44.178,158.523
C00921=1035.010,306.094,-121.943,171.517,44.180,158.524
C00922=1035.020,306.472,-121.995,171.523,44.181,158.525
C00923=1035.032,306.849,-122.045,171.530,44.183,158.526
C00924=1035.038,307.097,-122.078,171.534,44.184,158.526
C00925=1035.045,307.344,-122.112,171.538,44.185,158.527
C00926=1035.053,307.592,-122.145,171.543,44.186,158.528
C00927=1035.060,307.840,-122.178,171.547,44.187,158.528
C00928=1035.066,308.087,-122.212,171.552,44.188,158.529
C00929=1035.074,308.335,-122.246,171.555,44.190,158.530
C00930=1035.081,308.582,-122.279,171.560,44.191,158.530
C00931=1035.088,308.830,-122.312,171.565,44.192,158.531
C00932=1035.095,309.077,-122.345,171.569,44.193,158.532
C00933=1035.102,309.325,-122.379,171.573,44.194,158.532
C00934=1035.109,309.573,-122.413,171.578,44.195,158.533
C00935=1035.116,309.821,-122.446,171.582,44.196,158.534
C00936=1035.124,310.068,-122.479,171.587,44.197,158.534
C00937=1035.131,310.315,-122.513,171.590,44.198,158.535
C00938=1035.138,310.563,-122.547,171.595,44.199,158.535
C00939=1035.145,310.811,-122.580,171.600,44.201,158.536
C00940=1035.153,311.058,-122.614,171.604,44.202,158.537
C00941=1035.160,311.306,-122.647,171.609,44.203,158.538
C00942=1035.168,311.553,-122.681,171.613,44.204,158.538
C00943=1035.174,311.800,-122.715,171.617,44.206,158.539
C00944=1035.181,312.048,-122.749,171.622,44.207,158.540
C00945=1035.188,312.296,-122.783,171.627,44.208,158.540
C00946=1035.194,312.544,-122.817,171.631,44.209,158.541
C00947=1035.202,312.792,-122.851,171.636,44.211,158.542
C00948=1035.208,313.039,-122.885,171.639,44.212,158.542
C00949=1035.215,313.286,-122.920,171.644,44.214,158.543
C00950=1035.222,313.534,-122.954,171.649,44.215,158.544
C00951=1035.229,313.782,-122.988,171.653,44.217,158.545
C00952=1035.236,314.029,-123.022,171.658,44.218,158.545
C00953=1035.243,314.276,-123.056,171.663,44.219,158.546
C00954=1035.249,314.524,-123.090,171.667,44.221,158.547
C00955=1035.256,314.771,-123.124,171.671,44.222,158.547
C00956=1035.263,315.019,-123.159,171.676,44.223,158.548
C00957=1035.270,315.266,-123.193,171.680,44.224,158.549
C00958=1035.277,315.514,-123.228,171.685,44.226,158.550
C00959=1035.284,315.761,-123.262,171.690,44.228,158.551
C00960=1035.292,316.009,-123.296,171.694,44.229,158.551
C00961=1035.298,316.256,-123.331,171.699,44.231,158.552
C00962=1035.305,316.504,-123.365,171.704,44.232,158.553
C00963=1035.312,316.752,-123.399,171.708,44.233,158.553
C00964=1035.319,316.999,-123.434,171.713,44.234,158.554
C00965=1035.326,317.247,-123.468,171.718,44.236,158.555
C00966=1035.333,317.494,-123.503,171.721,44.237,158.556
C00967=1035.341,317.742,-123.537,171.726,44.239,158.556
C00968=1035.347,317.989,-123.572,171.731,44.240,158.557
C00969=1035.355,318.237,-123.606,171.736,44.241,158.558
C00970=1035.361,318.484,-123.641,171.740,44.243,158.559
C00971=1035.369,318.732,-123.675,171.745,44.245,158.559
C00972=1035.375,318.979,-123.710,171.750,44.246,158.560
C00973=1035.383,319.226,-123.744,171.755,44.247,158.561
C00974=1035.389,319.474,-123.779,171.759,44.249,158.562
C00975=1035.397,319.721,-123.813,171.764,44.250,158.562
C00976=1035.408,320.103,-123.867,171.771,44.253,158.564
C00977=1035.418,320.486,-123.920,171.779,44.255,158.565
C00978=1035.430,320.868,-123.973,171.786,44.257,158.566
C00979=1035.441,321.250,-124.027,171.792,44.260,158.567
C00980=1035.448,321.498,-124.062,171.797,44.261,158.568
C00981=1035.455,321.745,-124.096,171.802,44.263,158.569
C00982=1035.462,321.993,-124.131,171.807,44.264,158.569
C00983=1035.470,322.240,-124.166,171.812,44.265,158.570
C00984=1035.477,322.488,-124.201,171.816,44.267,158.571
C00985=1035.484,322.735,-124.235,171.821,44.269,158.572
C00986=1035.491,322.982,-124.271,171.826,44.270,158.573
C00987=1035.499,323.230,-124.306,171.831,44.272,158.574
C00988=1035.506,323.477,-124.341,171.836,44.273,158.574
C00989=1035.513,323.725,-124.374,171.841,44.275,158.575
C00990=1035.520,323.973,-124.410,171.846,44.276,158.576
C00991=1035.528,324.220,-124.445,171.850,44.278,158.577
C00992=1035.535,324.468,-124.480,171.855,44.280,158.577
C00993=1035.542,324.715,-124.514,171.860,44.281,158.578
C00994=1035.550,324.963,-124.550,171.865,44.283,158.579
C00995=1035.557,325.210,-124.584,171.870,44.284,158.580
C00996=1035.564,325.457,-124.619,171.875,44.285,158.581
C00997=1035.572,325.705,-124.654,171.880,44.287,158.581
C00998=1035.579,325.952,-124.689,171.885,44.289,158.582
C00999=1035.587,326.200,-124.724,171.889,44.290,158.583
C01000=1035.594,326.447,-124.759,171.894,44.292,158.584
C01001=1035.601,326.694,-124.794,171.899,44.294,158.585
C01002=1035.609,326.942,-124.830,171.904,44.295,158.586
C01003=1035.616,327.189,-124.865,171.909,44.297,158.586
C01004=1035.624,327.437,-124.900,171.914,44.298,158.587
C01005=1035.631,327.684,-124.935,171.919,44.300,158.588
C01006=1035.638,327.931,-124.970,171.924,44.302,158.589
C01007=1035.646,328.179,-125.005,171.929,44.303,158.590
C01008=1035.653,328.426,-125.041,171.934,44.305,158.591
C01009=1035.660,328.674,-125.076,171.939,44.307,158.592
C01010=1035.667,328.921,-125.111,171.944,44.309,158.592
C01011=1035.675,329.169,-125.148,171.949,44.310,158.593
C01012=1035.682,329.416,-125.183,171.953,44.313,158.594
C01013=1035.689,329.663,-125.219,171.958,44.314,158.595
C01014=1035.696,329.911,-125.254,171.963,44.316,158.596
C01015=1035.704,330.157,-125.289,171.968,44.317,158.597
C01016=1035.711,330.405,-125.325,171.974,44.320,158.598
C01017=1035.718,330.652,-125.361,171.979,44.321,158.598
C01018=1035.726,330.900,-125.396,171.984,44.323,158.599
C01019=1035.733,331.147,-125.432,171.989,44.325,158.600
C01020=1035.740,331.395,-125.467,171.994,44.326,158.601
C01021=1035.747,331.642,-125.503,171.999,44.328,158.602
C01022=1035.755,331.889,-125.540,172.004,44.330,158.603
C01023=1035.762,332.137,-125.575,172.009,44.332,158.604
C01024=1035.769,332.384,-125.611,172.014,44.334,158.605
C01025=1035.776,332.631,-125.647,172.019,44.336,158.606
C01026=1035.784,332.879,-125.682,172.025,44.338,158.607
C01027=1035.792,333.126,-125.718,172.030,44.339,158.607
C01028=1035.799,333.373,-125.754,172.035,44.341,158.608
C01029=1035.806,333.621,-125.790,172.040,44.343,158.609
C01030=1035.813,333.868,-125.826,172.045,44.345,158.610
C01031=1035.821,334.115,-125.862,172.050,44.347,158.611
C01032=1035.833,334.493,-125.917,172.058,44.350,158.613
C01033=1035.844,334.871,-125.972,172.066,44.353,158.614
C01034=1035.854,335.248,-126.027,172.073,44.356,158.615
C01035=1035.866,335.625,-126.082,172.082,44.359,158.617
C01036=1035.873,335.873,-126.119,172.088,44.361,158.618
C01037=1035.880,336.120,-126.155,172.093,44.362,158.619
C01038=1035.888,336.367,-126.191,172.098,44.365,158.620
C01039=1035.896,336.615,-126.227,172.103,44.367,158.621
C01040=1035.903,336.862,-126.263,172.108,44.368,158.622
C01041=1035.910,337.109,-126.300,172.113,44.370,158.623
C01042=1035.917,337.357,-126.336,172.119,44.373,158.624
C01043=1035.925,337.603,-126.372,172.124,44.375,158.625
C01044=1035.932,337.851,-126.408,172.129,44.377,158.626
C01045=1035.940,338.098,-126.444,172.134,44.379,158.626
C01046=1035.947,338.346,-126.481,172.139,44.381,158.627
C01047=1035.955,338.593,-126.518,172.146,44.383,158.628
C01048=1035.962,338.840,-126.554,172.151,44.385,158.629
C01049=1035.970,339.087,-126.590,172.156,44.387,158.630
C01050=1035.977,339.335,-126.627,172.161,44.389,158.631
C01051=1035.985,339.582,-126.664,172.166,44.391,158.632
C01052=1035.992,339.829,-126.700,172.172,44.393,158.633
C01053=1036.000,340.077,-126.736,172.177,44.395,158.634
C01054=1036.007,340.323,-126.773,172.183,44.397,158.635
C01055=1036.014,340.571,-126.810,172.189,44.399,158.636
C01056=1036.022,340.818,-126.846,172.194,44.401,158.637
C01057=1036.030,341.065,-126.883,172.199,44.404,158.638
C01058=1036.037,341.313,-126.920,172.204,44.406,158.639
C01059=1036.045,341.559,-126.957,172.210,44.408,158.640
C01060=1036.052,341.807,-126.993,172.216,44.410,158.641
C01061=1036.060,342.054,-127.030,172.221,44.412,158.642
C01062=1036.067,342.301,-127.067,172.226,44.414,158.643
C01063=1036.074,342.548,-127.104,172.232,44.416,158.644
C01064=1036.082,342.795,-127.140,172.237,44.419,158.646
C01065=1036.089,343.042,-127.177,172.242,44.421,158.647
C01066=1036.097,343.289,-127.214,172.249,44.423,158.648
C01067=1036.104,343.537,-127.251,172.254,44.425,158.649
C01068=1036.112,343.784,-127.288,172.259,44.427,158.650
C01069=1036.119,344.031,-127.326,172.265,44.430,158.651
C01070=1036.127,344.278,-127.363,172.271,44.432,158.652
C01071=1036.134,344.526,-127.399,172.276,44.434,158.653
C01072=1036.142,344.772,-127.436,172.282,44.437,158.654
C01073=1036.149,345.019,-127.474,172.287,44.439,158.655
C01074=1036.157,345.266,-127.511,172.293,44.441,158.656
C01075=1036.164,345.513,-127.548,172.299,44.443,158.657
C01076=1036.172,345.761,-127.585,172.304,44.446,158.658
C01077=1036.180,346.009,-127.622,172.309,44.448,158.659
C01078=1036.187,346.256,-127.660,172.316,44.450,158.660
C01079=1036.195,346.503,-127.697,172.321,44.453,158.661
C01080=1036.202,346.750,-127.734,172.327,44.455,158.662
C01081=1036.210,346.997,-127.771,172.332,44.458,158.664
C01082=1036.218,347.244,-127.809,172.338,44.460,158.665
C01083=1036.225,347.491,-127.846,172.344,44.463,158.666
C01084=1036.233,347.738,-127.883,172.349,44.465,158.667
C01085=1036.240,347.985,-127.921,172.356,44.467,158.668
C01086=1036.249,348.232,-127.958,172.361,44.469,158.669
C01087=1036.256,348.480,-127.996,172.366,44.472,158.670
C01088=1036.268,348.853,-128.053,172.375,44.475,158.672
C01089=1036.279,349.228,-128.110,172.384,44.479,158.673
C01090=1036.291,349.601,-128.167,172.393,44.483,158.675
C01091=1036.302,349.976,-128.223,172.402,44.487,158.677
C01092=1036.311,350.223,-128.261,172.407,44.489,158.678
C01093=1036.318,350.470,-128.299,172.413,44.492,158.679
C01094=1036.325,350.717,-128.336,172.419,44.494,158.680
C01095=1036.333,350.964,-128.375,172.425,44.496,158.681
C01096=1036.341,351.211,-128.413,172.431,44.499,158.683
C01097=1036.349,351.458,-128.450,172.437,44.501,158.684
C01098=1036.356,351.705,-128.488,172.442,44.504,158.685
C01099=1036.364,351.952,-128.526,172.449,44.507,158.686
C01100=1036.371,352.199,-128.564,172.454,44.509,158.687
C01101=1036.379,352.446,-128.602,172.461,44.511,158.689
C01102=1036.387,352.694,-128.640,172.466,44.514,158.690
C01103=1036.394,352.940,-128.678,172.472,44.517,158.691
C01104=1036.402,353.187,-128.715,172.478,44.519,158.692
C01105=1036.411,353.434,-128.754,172.484,44.522,158.693
C01106=1036.418,353.681,-128.792,172.490,44.525,158.695
C01107=1036.426,353.928,-128.830,172.496,44.527,158.696
C01108=1036.434,354.175,-128.868,172.502,44.530,158.697
C01109=1036.441,354.421,-128.906,172.508,44.533,158.698
C01110=1036.449,354.669,-128.944,172.514,44.535,158.699
C01111=1036.456,354.916,-128.983,172.520,44.538,158.700
C01112=1036.465,355.163,-129.021,172.527,44.540,158.702
C01113=1036.473,355.409,-129.059,172.532,44.543,158.703
C01114=1036.481,355.657,-129.097,172.539,44.545,158.704
C01115=1036.488,355.904,-129.135,172.544,44.548,158.705
C01116=1036.496,356.151,-129.174,172.551,44.551,158.707
C01117=1036.504,356.397,-129.212,172.556,44.554,158.708
C01118=1036.512,356.645,-129.250,172.563,44.556,158.709
C01119=1036.520,356.891,-129.289,172.569,44.559,158.710
C01120=1036.528,357.138,-129.327,172.575,44.562,158.712
C01121=1036.535,357.385,-129.366,172.581,44.565,158.713
C01122=1036.544,357.632,-129.404,172.587,44.567,158.714
C01123=1036.552,357.879,-129.443,172.593,44.570,158.715
C01124=1036.559,358.126,-129.482,172.600,44.573,158.717
C01125=1036.567,358.373,-129.520,172.606,44.576,158.718
C01126=1036.575,358.619,-129.559,172.612,44.578,158.719
C01127=1036.583,358.866,-129.598,172.619,44.582,158.720
C01128=1036.591,359.114,-129.636,172.624,44.584,158.722
C01129=1036.598,359.360,-129.675,172.631,44.587,158.723
C01130=1036.607,359.607,-129.713,172.638,44.590,158.724
C01131=1036.615,359.854,-129.753,172.643,44.593,158.726
C01132=1036.623,360.100,-129.791,172.650,44.596,158.727
C01133=1036.631,360.348,-129.829,172.656,44.599,158.728
C01134=1036.638,360.595,-129.869,172.662,44.601,158.729
C01135=1036.646,360.841,-129.908,172.669,44.604,158.731
C01136=1036.654,361.088,-129.946,172.675,44.607,158.732
C01137=1036.663,361.335,-129.985,172.681,44.610,158.733
C01138=1036.671,361.582,-130.024,172.688,44.613,158.735
C01139=1036.679,361.828,-130.063,172.694,44.616,158.736
C01140=1036.686,362.075,-130.102,172.701,44.619,158.737
C01141=1036.694,362.322,-130.142,172.707,44.622,158.739
C01142=1036.702,362.570,-130.181,172.713,44.625,158.740
C01143=1036.710,362.815,-130.220,172.720,44.628,158.741
C01144=1036.723,363.196,-130.281,172.730,44.633,158.744
C01145=1036.735,363.576,-130.341,172.740,44.637,158.746
C01146=1036.747,363.956,-130.402,172.750,44.642,158.748
C01147=1036.759,364.337,-130.462,172.760,44.647,158.750
C01148=1036.767,364.583,-130.501,172.767,44.650,158.751
C01149=1036.775,364.830,-130.541,172.773,44.653,158.753
C01150=1036.784,365.077,-130.581,172.779,44.656,158.754
C01151=1036.791,365.324,-130.620,172.786,44.659,158.756
C01152=1036.799,365.571,-130.659,172.793,44.663,158.757
C01153=1036.807,365.818,-130.699,172.800,44.666,158.758
C01154=1036.816,366.064,-130.738,172.805,44.669,158.760
C01155=1036.824,366.311,-130.778,172.812,44.672,158.761
C01156=1036.832,366.558,-130.818,172.819,44.675,158.762
C01157=1036.840,366.804,-130.857,172.826,44.678,158.764
C01158=1036.848,367.051,-130.897,172.833,44.681,158.765
C01159=1036.856,367.298,-130.936,172.840,44.684,158.767
C01160=1036.864,367.544,-130.977,172.846,44.688,158.768
C01161=1036.873,367.791,-131.016,172.852,44.691,158.770
C01162=1036.881,368.037,-131.055,172.859,44.694,158.771
C01163=1036.889,368.284,-131.095,172.866,44.697,158.772
C01164=1036.898,368.531,-131.135,172.873,44.701,158.774
C01165=1036.906,368.777,-131.175,172.880,44.704,158.775
C01166=1036.914,369.024,-131.215,172.887,44.707,158.777
C01167=1036.922,369.271,-131.255,172.894,44.710,158.778
C01168=1036.931,369.518,-131.294,172.900,44.714,158.780
C01169=1036.939,369.764,-131.335,172.906,44.717,158.781
C01170=1036.947,370.011,-131.374,172.914,44.720,158.783
C01171=1036.955,370.258,-131.414,172.920,44.723,158.784
C01172=1036.964,370.504,-131.454,172.927,44.727,158.786
C01173=1036.972,370.750,-131.495,172.934,44.730,158.787
C01174=1036.980,370.998,-131.535,172.941,44.734,158.789
C01175=1036.988,371.244,-131.576,172.948,44.737,158.790
C01176=1036.997,371.490,-131.615,172.955,44.740,158.792
C01177=1037.005,371.737,-131.656,172.962,44.744,158.793
C01178=1037.013,371.983,-131.696,172.969,44.747,158.795
C01179=1037.021,372.231,-131.737,172.976,44.750,158.796
C01180=1037.029,372.477,-131.777,172.983,44.754,158.798
C01181=1037.038,372.723,-131.817,172.990,44.758,158.800
C01182=1037.046,372.969,-131.858,172.998,44.761,158.801
C01183=1037.054,373.217,-131.898,173.005,44.765,158.803
C01184=1037.062,373.463,-131.939,173.011,44.768,158.804
C01185=1037.071,373.709,-131.979,173.019,44.771,158.806
C01186=1037.080,373.956,-132.020,173.026,44.775,158.807
C01187=1037.088,374.202,-132.061,173.033,44.779,158.809
C01188=1037.096,374.449,-132.101,173.040,44.782,158.810
C01189=1037.104,374.696,-132.142,173.047,44.786,158.812
C01190=1037.113,374.942,-132.182,173.054,44.789,158.814
C01191=1037.121,375.188,-132.223,173.061,44.793,158.815
C01192=1037.130,375.435,-132.264,173.068,44.797,158.817
C01193=1037.138,375.681,-132.304,173.075,44.800,158.818
C01194=1037.147,375.928,-132.345,173.082,44.804,158.820
C01195=1037.155,376.174,-132.385,173.090,44.807,158.822
C01196=1037.164,376.421,-132.426,173.098,44.811,158.823
C01197=1037.172,376.667,-132.467,173.105,44.814,158.825
C01198=1037.181,376.914,-132.509,173.112,44.818,158.826
C01199=1037.189,377.160,-132.549,173.119,44.822,158.828
C01200=1037.203,377.561,-132.615,173.132,44.828,158.831
C01201=1037.217,377.961,-132.682,173.143,44.834,158.834
C01202=1037.231,378.362,-132.749,173.155,44.840,158.836
C01203=1037.245,378.763,-132.816,173.167,44.846,158.839
C01204=1037.254,379.009,-132.857,173.174,44.850,158.841
C01205=1037.262,379.255,-132.898,173.182,44.854,158.842
C01206=1037.270,379.502,-132.940,173.189,44.857,158.844
C01207=1037.279,379.748,-132.982,173.197,44.861,158.846
C01208=1037.287,379.995,-133.023,173.204,44.865,158.847
C01209=1037.296,380.241,-133.064,173.212,44.869,158.849
C01210=1037.305,380.487,-133.106,173.219,44.873,158.851
C01211=1037.313,380.734,-133.147,173.227,44.876,158.852
C01212=1037.322,380.980,-133.189,173.235,44.881,158.854
C01213=1037.331,381.227,-133.230,173.242,44.885,158.856
C01214=1037.338,381.472,-133.272,173.250,44.889,158.858
C01215=1037.347,381.719,-133.314,173.258,44.892,158.859
C01216=1037.356,381.965,-133.356,173.265,44.896,158.861
C01217=1037.365,382.212,-133.397,173.273,44.900,158.863
C01218=1037.373,382.458,-133.438,173.281,44.904,158.865
C01219=1037.382,382.704,-133.480,173.288,44.908,158.867
C01220=1037.390,382.951,-133.522,173.296,44.912,158.868
C01221=1037.399,383.197,-133.564,173.304,44.916,158.870
C01222=1037.408,383.444,-133.605,173.311,44.920,158.872
C01223=1037.417,383.689,-133.648,173.319,44.924,158.874
C01224=1037.426,383.936,-133.690,173.327,44.929,158.876
C01225=1037.435,384.181,-133.731,173.335,44.932,158.877
C01226=1037.443,384.428,-133.773,173.343,44.937,158.879
C01227=1037.452,384.674,-133.815,173.350,44.941,158.881
C01228=1037.461,384.921,-133.857,173.358,44.945,158.883
C01229=1037.470,385.167,-133.899,173.366,44.949,158.885
C01230=1037.479,385.413,-133.941,173.374,44.953,158.886
C01231=1037.488,385.659,-133.983,173.382,44.957,158.888
C01232=1037.496,385.905,-134.026,173.390,44.961,158.890
C01233=1037.505,386.152,-134.067,173.398,44.965,158.892
C01234=1037.514,386.398,-134.109,173.406,44.969,158.894
C01235=1037.523,386.644,-134.151,173.414,44.974,158.896
C01236=1037.533,386.891,-134.194,173.422,44.978,158.898
C01237=1037.542,387.137,-134.236,173.430,44.982,158.899
C01238=1037.550,387.383,-134.278,173.438,44.986,158.901
C01239=1037.560,387.629,-134.321,173.447,44.990,158.903
C01240=1037.568,387.875,-134.362,173.454,44.995,158.905
C01241=1037.577,388.121,-134.405,173.463,44.999,158.907
C01242=1037.586,388.367,-134.448,173.470,45.003,158.909
C01243=1037.595,388.613,-134.491,173.479,45.007,158.911
C01244=1037.604,388.860,-134.533,173.486,45.012,158.913
C01245=1037.613,389.106,-134.575,173.495,45.016,158.915
C01246=1037.622,389.352,-134.618,173.504,45.021,158.917
C01247=1037.631,389.598,-134.661,173.511,45.025,158.919
C01248=1037.640,389.844,-134.704,173.520,45.029,158.921
C01249=1037.650,390.090,-134.747,173.529,45.034,158.923
C01250=1037.658,390.336,-134.790,173.536,45.038,158.925
C01251=1037.667,390.582,-134.832,173.545,45.043,158.927
C01252=1037.676,390.829,-134.876,173.554,45.047,158.929
C01253=1037.686,391.075,-134.918,173.561,45.052,158.930
C01254=1037.694,391.321,-134.961,173.570,45.056,158.933
C01255=1037.703,391.566,-135.003,173.579,45.060,158.935
C01256=1037.711,391.784,-135.043,173.586,45.065,158.936
C01257=1037.720,392.002,-135.080,173.593,45.069,158.938
C01258=1037.727,392.219,-135.118,173.601,45.072,158.940
C01259=1037.736,392.437,-135.156,173.608,45.076,158.942
C01260=1037.744,392.654,-135.195,173.615,45.080,158.943
C01261=1037.752,392.872,-135.233,173.623,45.085,158.945
C01262=1037.760,393.089,-135.271,173.631,45.089,158.947
C01263=1037.768,393.308,-135.309,173.639,45.093,158.949
C01264=1037.777,393.553,-135.352,173.647,45.097,158.951
C01265=1037.786,393.799,-135.396,173.655,45.102,158.953
C01266=1037.795,394.045,-135.439,173.664,45.107,158.955
C01267=1037.805,394.291,-135.482,173.673,45.111,158.957
C01268=1037.814,394.537,-135.526,173.682,45.116,158.959
C01269=1037.823,394.783,-135.570,173.691,45.120,158.961
C01270=1037.833,395.029,-135.613,173.700,45.125,158.964
C01271=1037.842,395.275,-135.657,173.707,45.130,158.966
C01272=1037.851,395.521,-135.701,173.716,45.135,158.968
C01273=1037.860,395.766,-135.745,173.725,45.139,158.970
C01274=1037.869,396.013,-135.788,173.734,45.144,158.972
C01275=1037.879,396.259,-135.831,173.743,45.149,158.974
C01276=1037.888,396.504,-135.875,173.752,45.154,158.976
C01277=1037.898,396.751,-135.919,173.761,45.158,158.978
C01278=1037.906,396.996,-135.963,173.770,45.163,158.981
C01279=1037.916,397.242,-136.007,173.779,45.168,158.983
C01280=1037.926,397.488,-136.051,173.788,45.173,158.985
C01281=1037.935,397.734,-136.095,173.797,45.178,158.987
C01282=1037.944,397.979,-136.138,173.806,45.183,158.989
C01283=1037.954,398.226,-136.183,173.815,45.188,158.992
C01284=1037.963,398.472,-136.227,173.824,45.193,158.994
C01285=1037.974,398.717,-136.271,173.833,45.198,158.996
C01286=1037.983,398.963,-136.315,173.842,45.203,158.998
C01287=1037.992,399.208,-136.359,173.851,45.208,159.000
C01288=1038.001,399.455,-136.403,173.859,45.213,159.003
C01289=1038.011,399.700,-136.448,173.869,45.218,159.005
C01290=1038.020,399.946,-136.492,173.879,45.223,159.007
C01291=1038.030,400.192,-136.536,173.888,45.228,159.010
C01292=1038.039,400.438,-136.581,173.897,45.233,159.012
C01293=1038.049,400.684,-136.625,173.906,45.238,159.014
C01294=1038.059,400.930,-136.670,173.915,45.243,159.016
C01295=1038.068,401.176,-136.714,173.924,45.248,159.019
C01296=1038.078,401.421,-136.759,173.934,45.253,159.021
C01297=1038.087,401.667,-136.803,173.944,45.258,159.023
C01298=1038.097,401.913,-136.848,173.953,45.263,159.026
C01299=1038.107,402.158,-136.892,173.962,45.269,159.028
C01300=1038.116,402.404,-136.937,173.971,45.274,159.030
C01301=1038.126,402.649,-136.982,173.981,45.279,159.033
C01302=1038.135,402.896,-137.026,173.990,45.284,159.035
C01303=1038.146,403.142,-137.071,174.000,45.290,159.037
C01304=1038.155,403.388,-137.117,174.010,45.295,159.040
C01305=1038.164,403.633,-137.162,174.019,45.300,159.042
C01306=1038.174,403.879,-137.206,174.029,45.306,159.045
C01307=1038.184,404.124,-137.251,174.039,45.311,159.047
C01308=1038.193,404.370,-137.297,174.048,45.316,159.050
C01309=1038.203,404.616,-137.343,174.057,45.322,159.052
C01310=1038.213,404.861,-137.387,174.068,45.327,159.054
C01311=1038.223,405.107,-137.432,174.077,45.332,159.057
C01312=1038.232,405.352,-137.478,174.086,45.338,159.059
C01313=1038.242,405.599,-137.523,174.097,45.344,159.062
C01314=1038.252,405.843,-137.568,174.106,45.349,159.064
C01315=1038.262,406.090,-137.614,174.117,45.354,159.067
C01316=1038.270,406.317,-137.656,174.126,45.360,159.069
C01317=1038.280,406.545,-137.698,174.135,45.364,159.071
C01318=1038.289,406.772,-137.740,174.144,45.370,159.074
C01319=1038.299,406.999,-137.782,174.153,45.375,159.076
C01320=1038.308,407.227,-137.824,174.163,45.380,159.078
C01321=1038.317,407.455,-137.866,174.172,45.385,159.081
C01322=1038.326,407.683,-137.909,174.181,45.390,159.083
C01323=1038.335,407.910,-137.951,174.190,45.396,159.086
C01324=1038.345,408.156,-137.997,174.201,45.401,159.088
C01325=1038.355,408.401,-138.042,174.210,45.407,159.091
C01326=1038.365,408.647,-138.089,174.221,45.412,159.093
C01327=1038.375,408.892,-138.134,174.230,45.418,159.096
C01328=1038.386,409.138,-138.179,174.241,45.424,159.098
C01329=1038.396,409.384,-138.226,174.251,45.429,159.101
C01330=1038.406,409.629,-138.271,174.261,45.435,159.104
C01331=1038.416,409.874,-138.317,174.272,45.441,159.106
C01332=1038.426,410.120,-138.364,174.282,45.447,159.109
C01333=1038.437,410.366,-138.410,174.293,45.452,159.111
C01334=1038.447,410.611,-138.455,174.302,45.458,159.114
C01335=1038.457,410.857,-138.502,174.313,45.464,159.117
C01336=1038.467,411.102,-138.548,174.324,45.469,159.119
C01337=1038.478,411.348,-138.594,174.335,45.476,159.122
C01338=1038.488,411.594,-138.640,174.344,45.482,159.125
C01339=1038.499,411.839,-138.687,174.355,45.487,159.128
C01340=1038.508,412.084,-138.733,174.366,45.494,159.130
C01341=1038.518,412.330,-138.779,174.376,45.499,159.133
C01342=1038.529,412.575,-138.826,174.387,45.505,159.136
C01343=1038.539,412.821,-138.873,174.398,45.511,159.139
C01344=1038.549,413.066,-138.920,174.409,45.517,159.141
C01345=1038.560,413.312,-138.966,174.418,45.523,159.144
C01346=1038.570,413.557,-139.013,174.429,45.529,159.147
C01347=1038.580,413.802,-139.060,174.440,45.536,159.150
C01348=1038.591,414.048,-139.106,174.451,45.542,159.153
C01349=1038.601,414.293,-139.153,174.462,45.548,159.155
C01350=1038.612,414.538,-139.200,174.473,45.554,159.158
C01351=1038.622,414.784,-139.246,174.484,45.560,159.161
C01352=1038.632,415.029,-139.294,174.495,45.566,159.164
C01353=1038.643,415.274,-139.340,174.506,45.572,159.167
C01354=1038.653,415.520,-139.388,174.517,45.578,159.169
C01355=1038.664,415.765,-139.435,174.529,45.585,159.173
C01356=1038.675,416.010,-139.482,174.540,45.591,159.175
C01357=1038.685,416.256,-139.529,174.551,45.597,159.178
C01358=1038.695,416.501,-139.576,174.561,45.603,159.181
C01359=1038.706,416.747,-139.623,174.573,45.610,159.184
C01360=1038.717,416.992,-139.670,174.584,45.616,159.187
C01361=1038.727,417.237,-139.718,174.596,45.622,159.190
C01362=1038.738,417.483,-139.766,174.607,45.629,159.193
C01363=1038.749,417.728,-139.812,174.618,45.635,159.196
C01364=1038.759,417.972,-139.860,174.629,45.641,159.199
C01365=1038.770,418.218,-139.908,174.641,45.648,159.202
C01366=1038.780,418.464,-139.955,174.652,45.654,159.205
C01367=1038.791,418.709,-140.003,174.663,45.661,159.208
C01368=1038.802,418.954,-140.051,174.676,45.667,159.211
C01369=1038.812,419.199,-140.099,174.687,45.674,159.214
C01370=1038.823,419.444,-140.147,174.698,45.680,159.217
C01371=1038.834,419.689,-140.195,174.710,45.687,159.220
C01372=1038.845,419.935,-140.242,174.722,45.694,159.223
C01373=1038.856,420.180,-140.291,174.733,45.700,159.226
C01374=1038.866,420.425,-140.339,174.745,45.707,159.229
C01375=1038.877,420.670,-140.387,174.757,45.713,159.232
C01376=1038.887,420.890,-140.430,174.768,45.719,159.235
C01377=1038.897,421.111,-140.473,174.779,45.725,159.238
C01378=1038.906,421.331,-140.516,174.789,45.731,159.241
C01379=1038.917,421.551,-140.560,174.799,45.737,159.244
C01380=1038.927,421.772,-140.603,174.810,45.743,159.247
C01381=1038.936,421.992,-140.646,174.821,45.749,159.250
C01382=1038.946,422.212,-140.690,174.832,45.755,159.252
C01383=1038.956,422.432,-140.733,174.843,45.761,159.255
C01384=1038.967,422.678,-140.781,174.855,45.769,159.259
C01385=1038.978,422.922,-140.830,174.867,45.775,159.262
C01386=1038.989,423.168,-140.878,174.880,45.782,159.265
C01387=1039.001,423.413,-140.927,174.892,45.789,159.268
C01388=1039.012,423.658,-140.976,174.904,45.796,159.272
C01389=1039.023,423.903,-141.024,174.916,45.803,159.275
C01390=1039.034,424.148,-141.073,174.929,45.810,159.278
C01391=1039.046,424.393,-141.122,174.942,45.817,159.281
C01392=1039.057,424.638,-141.170,174.953,45.824,159.285
C01393=1039.068,424.883,-141.220,174.966,45.831,159.288
C01394=1039.079,425.128,-141.269,174.978,45.837,159.291
C01395=1039.090,425.373,-141.318,174.991,45.845,159.295
C01396=1039.102,425.618,-141.366,175.004,45.852,159.298
C01397=1039.113,425.863,-141.415,175.016,45.859,159.302
C01398=1039.124,426.108,-141.465,175.029,45.866,159.305
C01399=1039.135,426.352,-141.514,175.042,45.873,159.308
C01400=1039.146,426.597,-141.563,175.055,45.880,159.312
C01401=1039.158,426.842,-141.612,175.068,45.888,159.315
C01402=1039.170,427.087,-141.662,175.080,45.894,159.319
C01403=1039.181,427.332,-141.712,175.093,45.902,159.322
C01404=1039.192,427.577,-141.761,175.106,45.909,159.326
C01405=1039.204,427.822,-141.810,175.119,45.916,159.329
C01406=1039.216,428.066,-141.860,175.132,45.924,159.333
C01407=1039.227,428.311,-141.909,175.145,45.931,159.336
C01408=1039.239,428.556,-141.959,175.159,45.938,159.340
C01409=1039.250,428.801,-142.009,175.172,45.946,159.343
C01410=1039.261,429.045,-142.059,175.185,45.953,159.347
C01411=1039.273,429.291,-142.109,175.198,45.961,159.351
C01412=1039.284,429.535,-142.158,175.211,45.968,159.354
C01413=1039.295,429.779,-142.209,175.225,45.976,159.358
C01414=1039.308,430.024,-142.259,175.238,45.983,159.361
C01415=1039.319,430.268,-142.309,175.251,45.991,159.365
C01416=1039.332,430.536,-142.363,175.267,45.999,159.369
C01417=1039.344,430.805,-142.419,175.281,46.007,159.373
C01418=1039.358,431.071,-142.473,175.296,46.016,159.377
C01419=1039.370,431.339,-142.528,175.311,46.024,159.381
C01420=1039.382,431.584,-142.578,175.325,46.031,159.385
C01421=1039.394,431.828,-142.629,175.338,46.039,159.389
C01422=1039.406,432.072,-142.679,175.353,46.047,159.392
C01423=1039.418,432.318,-142.730,175.366,46.055,159.396
C01424=1039.429,432.562,-142.780,175.380,46.062,159.400
C01425=1039.441,432.806,-142.831,175.395,46.070,159.404
C01426=1039.454,433.051,-142.881,175.408,46.078,159.408
C01427=1039.465,433.295,-142.933,175.422,46.085,159.411
C01428=1039.478,433.540,-142.983,175.437,46.093,159.415
C01429=1039.490,433.785,-143.034,175.450,46.101,159.419
C01430=1039.502,434.029,-143.085,175.465,46.109,159.423
C01431=1039.514,434.273,-143.135,175.479,46.117,159.427
C01432=1039.526,434.518,-143.187,175.494,46.125,159.431
C01433=1039.539,434.763,-143.237,175.508,46.133,159.435
C01434=1039.551,435.007,-143.289,175.522,46.141,159.439
C01435=1039.563,435.252,-143.340,175.536,46.149,159.443
C01436=1039.575,435.489,-143.389,175.551,46.157,159.447
C01437=1039.586,435.726,-143.439,175.565,46.165,159.451
C01438=1039.599,435.964,-143.489,175.579,46.172,159.454
C01439=1039.610,436.201,-143.539,175.593,46.180,159.458
C01440=1039.622,436.439,-143.589,175.608,46.188,159.462
C01441=1039.634,436.676,-143.639,175.623,46.196,159.466
C01442=1039.646,436.912,-143.689,175.637,46.204,159.470
C01443=1039.658,437.151,-143.739,175.650,46.212,159.474
C01444=1039.671,437.394,-143.791,175.666,46.220,159.478
C01445=1039.683,437.639,-143.842,175.681,46.229,159.483
C01446=1039.695,437.884,-143.895,175.696,46.237,159.487
C01447=1039.708,438.127,-143.946,175.711,46.245,159.491
C01448=1039.720,438.372,-143.998,175.726,46.254,159.495
C01449=1039.733,438.616,-144.050,175.742,46.262,159.499
C01450=1039.745,438.860,-144.102,175.757,46.270,159.503
C01451=1039.758,439.105,-144.155,175.772,46.279,159.508
C01452=1039.771,439.348,-144.206,175.788,46.287,159.512
C01453=1039.784,439.593,-144.259,175.803,46.296,159.516
C01454=1039.796,439.837,-144.311,175.819,46.304,159.521
C01455=1039.809,440.081,-144.363,175.834,46.313,159.525
C01456=1039.821,440.326,-144.416,175.850,46.321,159.529
C01457=1039.834,440.569,-144.467,175.866,46.330,159.534
C01458=1039.847,440.813,-144.521,175.882,46.339,159.538
C01459=1039.860,441.057,-144.573,175.897,46.347,159.542
C01460=1039.873,441.301,-144.626,175.913,46.356,159.547
C01461=1039.885,441.546,-144.678,175.929,46.364,159.551
C01462=1039.899,441.790,-144.732,175.945,46.373,159.556
C01463=1039.911,442.034,-144.784,175.961,46.382,159.560
C01464=1039.924,442.278,-144.837,175.977,46.390,159.565
C01465=1039.937,442.522,-144.890,175.994,46.400,159.569
C01466=1039.950,442.766,-144.943,176.009,46.408,159.574
C01467=1039.963,443.010,-144.996,176.026,46.417,159.578
C01468=1039.976,443.254,-145.049,176.042,46.426,159.583
C01469=1039.990,443.498,-145.102,176.059,46.435,159.588
C01470=1040.003,443.742,-145.155,176.075,46.444,159.592
C01471=1040.016,443.986,-145.208,176.092,46.453,159.597
C01472=1040.029,444.228,-145.262,176.109,46.462,159.601
C01473=1040.042,444.472,-145.316,176.125,46.471,159.606
C01474=1040.056,444.715,-145.368,176.142,46.480,159.611
C01475=1040.070,444.959,-145.421,176.159,46.488,159.615
C01476=1040.085,445.202,-145.474,176.176,46.497,159.620
C01477=1040.100,445.445,-145.525,176.192,46.506,159.625
C01478=1040.115,445.688,-145.576,176.210,46.515,159.629
C01479=1040.131,445.934,-145.627,176.227,46.523,159.634
C01480=1040.148,446.176,-145.677,176.244,46.532,159.638
C01481=1040.166,446.420,-145.728,176.261,46.540,159.643
C01482=1040.183,446.664,-145.777,176.279,46.548,159.648
C01483=1040.202,446.909,-145.826,176.296,46.556,159.652
C01484=1040.221,447.152,-145.874,176.314,46.564,159.657
C01485=1040.242,447.397,-145.922,176.331,46.572,159.661
C01486=1040.261,447.641,-145.970,176.349,46.580,159.665
C01487=1040.282,447.886,-146.018,176.367,46.587,159.670
C01488=1040.304,448.130,-146.064,176.385,46.595,159.674
C01489=1040.326,448.374,-146.110,176.402,46.602,159.679
C01490=1040.349,448.619,-146.156,176.420,46.610,159.683
C01491=1040.372,448.864,-146.202,176.439,46.617,159.688
C01492=1040.395,449.110,-146.246,176.457,46.624,159.692
C01493=1040.420,449.354,-146.290,176.476,46.631,159.697
C01494=1040.445,449.599,-146.334,176.493,46.638,159.701
C01495=1040.470,449.845,-146.378,176.512,46.645,159.705
C01496=1040.496,450.081,-146.419,176.530,46.651,159.709
C01497=1040.521,450.317,-146.460,176.548,46.658,159.713
C01498=1040.547,450.554,-146.501,176.566,46.665,159.718
C01499=1040.575,450.790,-146.541,176.584,46.670,159.722
C01500=1040.602,451.026,-146.580,176.602,46.677,159.726
C01501=1040.629,451.262,-146.620,176.620,46.683,159.730
C01502=1040.658,451.498,-146.658,176.638,46.689,159.734
C01503=1040.686,451.732,-146.697,176.656,46.695,159.738
C01504=1040.390,451.779,-147.014,176.659,46.771,159.761
C01505=1040.362,451.552,-146.978,176.642,46.765,159.757
C01506=1040.334,451.323,-146.940,176.623,46.760,159.753
C01507=1040.307,451.095,-146.903,176.606,46.754,159.749
C01508=1040.281,450.866,-146.864,176.588,46.748,159.745
C01509=1040.255,450.638,-146.825,176.571,46.742,159.741
C01510=1040.228,450.409,-146.787,176.553,46.736,159.737
C01511=1040.204,450.180,-146.748,176.536,46.730,159.733
C01512=1040.179,449.951,-146.707,176.519,46.723,159.729
C01513=1040.153,449.706,-146.664,176.500,46.716,159.725
C01514=1040.128,449.461,-146.620,176.482,46.710,159.721
C01515=1040.103,449.216,-146.577,176.464,46.703,159.716
C01516=1040.079,448.971,-146.532,176.445,46.696,159.712
C01517=1040.055,448.726,-146.486,176.427,46.689,159.708
C01518=1040.032,448.482,-146.441,176.408,46.682,159.703
C01519=1040.010,448.237,-146.395,176.390,46.674,159.699
C01520=1039.988,447.992,-146.348,176.373,46.666,159.694
C01521=1039.967,447.747,-146.302,176.355,46.659,159.690
C01522=1039.946,447.503,-146.254,176.336,46.651,159.685
C01523=1039.926,447.259,-146.207,176.319,46.644,159.681
C01524=1039.907,447.015,-146.158,176.302,46.636,159.676
C01525=1039.888,446.771,-146.109,176.284,46.628,159.672
C01526=1039.870,446.527,-146.060,176.266,46.620,159.667
C01527=1039.851,446.282,-146.010,176.249,46.612,159.663
C01528=1039.835,446.039,-145.961,176.231,46.603,159.658
C01529=1039.818,445.795,-145.910,176.215,46.595,159.654
C01530=1039.801,445.551,-145.859,176.198,46.587,159.649
C01531=1039.786,445.308,-145.807,176.180,46.578,159.644
C01532=1039.771,445.065,-145.755,176.164,46.570,159.640
C01533=1039.757,444.821,-145.703,176.147,46.561,159.635
C01534=1039.744,444.578,-145.650,176.129,46.552,159.631
C01535=1039.729,444.334,-145.597,176.113,46.543,159.626
C01536=1039.717,444.092,-145.543,176.096,46.534,159.621
C01537=1039.704,443.848,-145.490,176.079,46.525,159.617
C01538=1039.690,443.604,-145.437,176.063,46.517,159.612
C01539=1039.677,443.360,-145.384,176.046,46.508,159.607
C01540=1039.663,443.116,-145.331,176.030,46.499,159.603
C01541=1039.650,442.872,-145.278,176.013,46.490,159.598
C01542=1039.637,442.628,-145.224,175.997,46.481,159.594
C01543=1039.625,442.384,-145.172,175.981,46.473,159.589
C01544=1039.611,442.140,-145.119,175.965,46.464,159.585
C01545=1039.598,441.896,-145.066,175.949,46.455,159.580
C01546=1039.586,441.653,-145.013,175.933,46.447,159.576
C01547=1039.573,441.408,-144.960,175.916,46.438,159.571
C01548=1039.560,441.164,-144.907,175.901,46.429,159.567
C01549=1039.546,440.920,-144.855,175.884,46.421,159.562
C01550=1039.534,440.676,-144.803,175.868,46.412,159.558
C01551=1039.521,440.432,-144.750,175.853,46.404,159.554
C01552=1039.508,440.187,-144.697,175.837,46.395,159.549
C01553=1039.496,439.943,-144.645,175.822,46.386,159.545
C01554=1039.483,439.699,-144.593,175.806,46.378,159.541
C01555=1039.470,439.455,-144.541,175.791,46.370,159.536
C01556=1039.458,439.211,-144.489,175.775,46.362,159.532
C01557=1039.445,438.967,-144.437,175.760,46.353,159.528
C01558=1039.433,438.722,-144.384,175.744,46.345,159.524
C01559=1039.420,438.478,-144.332,175.729,46.337,159.519
C01560=1039.407,438.234,-144.280,175.714,46.328,159.515
C01561=1039.395,437.990,-144.228,175.698,46.320,159.511
C01562=1039.383,437.746,-144.177,175.683,46.312,159.507
C01563=1039.370,437.501,-144.124,175.668,46.304,159.503
C01564=1039.357,437.257,-144.073,175.653,46.295,159.498
C01565=1039.346,437.019,-144.022,175.639,46.287,159.494
C01566=1039.334,436.781,-143.972,175.624,46.279,159.490
C01567=1039.322,436.543,-143.922,175.609,46.272,159.487
C01568=1039.310,436.305,-143.872,175.595,46.264,159.483
C01569=1039.297,436.067,-143.822,175.580,46.256,159.479
C01570=1039.285,435.829,-143.772,175.566,46.248,159.475
C01571=1039.273,435.591,-143.722,175.552,46.240,159.471
C01572=1039.261,435.353,-143.672,175.538,46.232,159.467
C01573=1039.250,435.108,-143.620,175.523,46.225,159.463
C01574=1039.238,434.864,-143.569,175.509,46.217,159.459
C01575=1039.225,434.620,-143.518,175.494,46.209,159.455
C01576=1039.213,434.374,-143.467,175.479,46.201,159.451
C01577=1039.201,434.130,-143.417,175.465,46.193,159.447
C01578=1039.189,433.886,-143.365,175.451,46.185,159.443
C01579=1039.176,433.641,-143.314,175.437,46.178,159.439
C01580=1039.164,433.397,-143.264,175.422,46.170,159.435
C01581=1039.152,433.152,-143.213,175.408,46.162,159.432
C01582=1039.140,432.907,-143.163,175.395,46.154,159.428
C01583=1039.128,432.663,-143.111,175.380,46.147,159.424
C01584=1039.116,432.419,-143.062,175.366,46.139,159.420
C01585=1039.105,432.174,-143.011,175.353,46.131,159.416
C01586=1039.092,431.929,-142.960,175.339,46.124,159.413
C01587=1039.080,431.684,-142.910,175.324,46.116,159.409
C01588=1039.069,431.440,-142.860,175.311,46.109,159.405
C01589=1039.056,431.195,-142.810,175.297,46.101,159.401
C01590=1039.045,430.950,-142.759,175.283,46.093,159.398
C01591=1039.033,430.706,-142.709,175.269,46.086,159.394
C01592=1039.022,430.461,-142.659,175.256,46.078,159.390
C01593=1039.010,430.217,-142.609,175.243,46.071,159.387
C01594=1038.998,429.972,-142.558,175.229,46.063,159.383
C01595=1038.987,429.728,-142.508,175.216,46.056,159.379
C01596=1038.975,429.482,-142.458,175.203,46.048,159.376
C01597=1038.964,429.238,-142.409,175.189,46.041,159.372
C01598=1038.951,428.993,-142.359,175.176,46.034,159.369
C01599=1038.940,428.748,-142.308,175.163,46.027,159.365
C01600=1038.929,428.504,-142.259,175.149,46.020,159.361
C01601=1038.917,428.258,-142.209,175.136,46.012,159.358
C01602=1038.906,428.014,-142.160,175.123,46.005,159.354
C01603=1038.894,427.770,-142.110,175.110,45.998,159.351
C01604=1038.883,427.524,-142.060,175.097,45.990,159.347
C01605=1038.872,427.279,-142.011,175.084,45.983,159.344
C01606=1038.860,427.034,-141.962,175.070,45.976,159.340
C01607=1038.848,426.790,-141.912,175.057,45.969,159.337
C01608=1038.837,426.545,-141.862,175.044,45.962,159.333
C01609=1038.826,426.300,-141.813,175.032,45.955,159.330
C01610=1038.814,426.055,-141.764,175.019,45.947,159.326
C01611=1038.803,425.810,-141.715,175.006,45.940,159.323
C01612=1038.792,425.566,-141.666,174.994,45.934,159.320
C01613=1038.780,425.321,-141.617,174.981,45.926,159.316
C01614=1038.770,425.075,-141.568,174.969,45.919,159.313
C01615=1038.758,424.830,-141.519,174.956,45.912,159.310
C01616=1038.747,424.586,-141.470,174.944,45.905,159.306
C01617=1038.736,424.356,-141.424,174.931,45.899,159.303
C01618=1038.726,424.127,-141.378,174.920,45.893,159.300
C01619=1038.716,423.897,-141.333,174.909,45.886,159.297
C01620=1038.705,423.667,-141.287,174.896,45.880,159.294
C01621=1038.694,423.437,-141.241,174.885,45.873,159.291
C01622=1038.684,423.208,-141.196,174.874,45.867,159.288
C01623=1038.673,422.977,-141.151,174.863,45.860,159.285
C01624=1038.663,422.748,-141.105,174.850,45.854,159.282
C01625=1038.652,422.503,-141.057,174.839,45.848,159.279
C01626=1038.641,422.258,-141.009,174.826,45.841,159.275
C01627=1038.630,422.013,-140.961,174.814,45.834,159.272
C01628=1038.619,421.768,-140.912,174.803,45.827,159.269
C01629=1038.608,421.516,-140.862,174.790,45.821,159.266
C01630=1038.596,421.265,-140.813,174.778,45.814,159.262
C01631=1038.585,421.014,-140.764,174.765,45.807,159.259
C01632=1038.574,420.762,-140.714,174.754,45.800,159.256
C01633=1038.563,420.517,-140.666,174.742,45.794,159.253
C01634=1038.552,420.272,-140.618,174.730,45.787,159.250
C01635=1038.541,420.027,-140.570,174.718,45.781,159.247
C01636=1038.531,419.782,-140.522,174.707,45.774,159.244
C01637=1038.520,419.536,-140.474,174.694,45.768,159.241
C01638=1038.509,419.292,-140.427,174.683,45.761,159.237
C01639=1038.498,419.047,-140.379,174.671,45.755,159.234
C01640=1038.487,418.801,-140.331,174.660,45.748,159.231
C01641=1038.476,418.556,-140.283,174.648,45.741,159.228
C01642=1038.466,418.311,-140.236,174.636,45.736,159.225
C01643=1038.455,418.065,-140.188,174.625,45.729,159.222
C01644=1038.445,417.820,-140.140,174.614,45.723,159.219
C01645=1038.434,417.575,-140.092,174.602,45.716,159.216
C01646=1038.424,417.329,-140.045,174.591,45.710,159.213
C01647=1038.413,417.085,-139.998,174.579,45.704,159.210
C01648=1038.402,416.839,-139.951,174.568,45.697,159.207
C01649=1038.392,416.593,-139.903,174.557,45.692,159.204
C01650=1038.381,416.348,-139.857,174.546,45.685,159.202
C01651=1038.371,416.103,-139.810,174.534,45.679,159.199
C01652=1038.359,415.858,-139.761,174.523,45.673,159.196
C01653=1038.349,415.613,-139.715,174.512,45.666,159.193
C01654=1038.339,415.367,-139.668,174.501,45.660,159.190
C01655=1038.328,415.121,-139.621,174.489,45.654,159.187
C01656=1038.318,414.876,-139.574,174.478,45.648,159.184
C01657=1038.307,414.630,-139.527,174.468,45.643,159.182
C01658=1038.297,414.385,-139.479,174.457,45.636,159.179
C01659=1038.286,414.140,-139.433,174.446,45.630,159.176
C01660=1038.276,413.894,-139.386,174.435,45.624,159.173
C01661=1038.266,413.649,-139.339,174.424,45.618,159.170
C01662=1038.255,413.404,-139.293,174.413,45.612,159.167
C01663=1038.245,413.158,-139.246,174.402,45.606,159.165
C01664=1038.234,412.913,-139.199,174.392,45.600,159.162
C01665=1038.224,412.667,-139.153,174.381,45.594,159.159
C01666=1038.214,412.423,-139.106,174.371,45.588,159.156
C01667=1038.204,412.177,-139.060,174.360,45.582,159.154
C01668=1038.194,411.932,-139.013,174.350,45.576,159.151
C01669=1038.184,411.686,-138.966,174.339,45.571,159.148
C01670=1038.173,411.440,-138.921,174.328,45.565,159.145
C01671=1038.163,411.194,-138.874,174.317,45.559,159.143
C01672=1038.153,410.949,-138.828,174.307,45.553,159.140
C01673=1038.142,410.703,-138.782,174.297,45.547,159.137
C01674=1038.133,410.458,-138.736,174.286,45.542,159.135
C01675=1038.122,410.212,-138.690,174.276,45.536,159.132
C01676=1038.111,409.967,-138.644,174.265,45.530,159.129
C01677=1038.101,409.721,-138.598,174.255,45.524,159.127
C01678=1038.091,409.476,-138.552,174.245,45.519,159.124
C01679=1038.081,409.230,-138.506,174.234,45.514,159.122
C01680=1038.070,408.985,-138.460,174.224,45.508,159.119
C01681=1038.061,408.740,-138.414,174.214,45.502,159.116
C01682=1038.050,408.494,-138.368,174.204,45.496,159.114
C01683=1038.040,408.248,-138.323,174.193,45.491,159.111
C01684=1038.031,408.003,-138.277,174.184,45.485,159.109
C01685=1038.021,407.774,-138.235,174.175,45.480,159.106
C01686=1038.012,407.546,-138.192,174.164,45.475,159.104
C01687=1038.002,407.317,-138.150,174.155,45.470,159.101
C01688=1037.993,407.088,-138.107,174.146,45.465,159.099
C01689=1037.984,406.860,-138.065,174.136,45.460,159.097
C01690=1037.975,406.631,-138.023,174.127,45.455,159.095
C01691=1037.965,406.402,-137.981,174.118,45.450,159.092
C01692=1037.956,406.174,-137.938,174.109,45.445,159.090
C01693=1037.946,405.928,-137.893,174.099,45.440,159.087
C01694=1037.937,405.682,-137.848,174.089,45.434,159.085
C01695=1037.927,405.437,-137.802,174.080,45.428,159.082
C01696=1037.917,405.191,-137.757,174.069,45.423,159.080
C01697=1037.907,404.946,-137.712,174.060,45.418,159.077
C01698=1037.898,404.699,-137.666,174.050,45.412,159.075
C01699=1037.888,404.454,-137.621,174.040,45.407,159.073
C01700=1037.878,404.209,-137.576,174.030,45.402,159.070
C01701=1037.868,403.963,-137.531,174.021,45.396,159.068
C01702=1037.859,403.717,-137.486,174.012,45.391,159.065
C01703=1037.849,403.471,-137.440,174.001,45.386,159.063
C01704=1037.839,403.226,-137.396,173.992,45.380,159.060
C01705=1037.829,402.980,-137.351,173.983,45.376,159.058
C01706=1037.820,402.735,-137.306,173.973,45.370,159.056
C01707=1037.811,402.488,-137.261,173.963,45.365,159.053
C01708=1037.801,402.243,-137.216,173.954,45.360,159.051
C01709=1037.791,401.996,-137.171,173.945,45.355,159.049
C01710=1037.781,401.751,-137.126,173.935,45.350,159.046
C01711=1037.772,401.505,-137.082,173.926,45.345,159.044
C01712=1037.762,401.259,-137.037,173.917,45.340,159.042
C01713=1037.752,401.014,-136.993,173.907,45.334,159.039
C01714=1037.743,400.768,-136.949,173.897,45.330,159.037
C01715=1037.733,400.522,-136.904,173.888,45.324,159.035
C01716=1037.724,400.276,-136.860,173.879,45.319,159.032
C01717=1037.714,400.031,-136.815,173.870,45.314,159.030
C01718=1037.705,399.785,-136.771,173.861,45.309,159.028
C01719=1037.696,399.539,-136.727,173.852,45.305,159.026
C01720=1037.686,399.293,-136.682,173.842,45.299,159.023
C01721=1037.676,399.048,-136.639,173.833,45.294,159.021
C01722=1037.667,398.801,-136.594,173.824,45.289,159.019
C01723=1037.657,398.555,-136.550,173.814,45.285,159.017
C01724=1037.648,398.310,-136.506,173.805,45.280,159.014
C01725=1037.639,398.064,-136.462,173.796,45.275,159.012
C01726=1037.629,397.819,-136.418,173.788,45.270,159.010
C01727=1037.619,397.572,-136.374,173.779,45.266,159.008
C01728=1037.610,397.326,-136.330,173.770,45.261,159.006
C01729=1037.601,397.081,-136.286,173.761,45.256,159.004
C01730=1037.592,396.835,-136.242,173.752,45.251,159.001
C01731=1037.581,396.589,-136.199,173.743,45.246,158.999
C01732=1037.573,396.343,-136.155,173.734,45.241,158.997
C01733=1037.563,396.097,-136.111,173.725,45.237,158.995
C01734=1037.554,395.851,-136.067,173.716,45.232,158.993
C01735=1037.545,395.605,-136.024,173.707,45.227,158.991
C01736=1037.535,395.359,-135.980,173.698,45.222,158.988
C01737=1037.526,395.114,-135.936,173.690,45.218,158.986
C01738=1037.517,394.868,-135.892,173.681,45.213,158.984
C01739=1037.508,394.621,-135.849,173.672,45.209,158.982
C01740=1037.498,394.376,-135.806,173.663,45.204,158.980
C01741=1037.489,394.129,-135.762,173.654,45.199,158.978
C01742=1037.480,393.884,-135.719,173.645,45.195,158.976
C01743=1037.471,393.637,-135.676,173.638,45.190,158.974
C01744=1037.462,393.392,-135.632,173.629,45.185,158.972
C01745=1037.453,393.173,-135.593,173.621,45.181,158.970
C01746=1037.445,392.955,-135.556,173.613,45.178,158.968
C01747=1037.437,392.736,-135.517,173.605,45.173,158.966
C01748=1037.428,392.517,-135.479,173.598,45.169,158.964
C01749=1037.421,392.299,-135.440,173.591,45.165,158.963
C01750=1037.412,392.080,-135.401,173.583,45.161,158.961
C01751=1037.405,391.861,-135.364,173.576,45.157,158.959
C01752=1037.396,391.643,-135.326,173.568,45.153,158.957
C01753=1037.387,391.396,-135.282,173.560,45.149,158.955
C01754=1037.379,391.150,-135.239,173.551,45.144,158.953
C01755=1037.369,390.905,-135.196,173.542,45.141,158.951
C01756=1037.360,390.659,-135.153,173.535,45.136,158.949
C01757=1037.351,390.413,-135.110,173.526,45.132,158.947
C01758=1037.342,390.167,-135.067,173.517,45.127,158.945
C01759=1037.333,389.920,-135.025,173.509,45.123,158.943
C01760=1037.324,389.674,-134.982,173.501,45.119,158.942
C01761=1037.315,389.428,-134.940,173.492,45.114,158.939
C01762=1037.306,389.182,-134.897,173.484,45.110,158.937
C01763=1037.297,388.935,-134.854,173.476,45.106,158.936
C01764=1037.288,388.690,-134.812,173.468,45.101,158.934
C01765=1037.279,388.444,-134.769,173.460,45.097,158.932
C01766=1037.270,388.198,-134.726,173.452,45.093,158.930
C01767=1037.262,387.951,-134.684,173.443,45.088,158.928
C01768=1037.252,387.705,-134.641,173.435,45.084,158.926
C01769=1037.243,387.460,-134.599,173.427,45.080,158.924
C01770=1037.234,387.213,-134.557,173.419,45.076,158.922
C01771=1037.225,386.967,-134.514,173.411,45.072,158.920
C01772=1037.216,386.720,-134.472,173.402,45.068,158.918
C01773=1037.207,386.474,-134.430,173.395,45.063,158.917
C01774=1037.198,386.228,-134.388,173.386,45.060,158.915
C01775=1037.189,385.982,-134.346,173.379,45.056,158.913
C01776=1037.181,385.736,-134.303,173.371,45.052,158.911
C01777=1037.172,385.489,-134.262,173.363,45.047,158.909
C01778=1037.163,385.243,-134.220,173.354,45.043,158.907
C01779=1037.153,384.997,-134.177,173.347,45.039,158.906
C01780=1037.145,384.751,-134.136,173.339,45.035,158.904
